LIN {X 0.008,Y -350.528,Z 1604.654,A 0.000,B 0.000,C 90.000,E1 117.719} C_DIS
LIN {X -0.132,Y -363.756,Z 1604.639,A 0.000,B 0.000,C 90.000,E1 115.027} C_DIS
LIN {X 0.133,Y -378.533,Z 1604.624,A 0.000,B 0.000,C 90.000,E1 112.333} C_DIS
LIN {X -0.125,Y -393.075,Z 1604.611,A 0.000,B 0.000,C 90.000,E1 110.066} C_DIS
LIN {X -0.167,Y -409.046,Z 1604.599,A 0.000,B 0.000,C 90.000,E1 107.819} C_DIS
LIN {X -0.066,Y -426.554,Z 1604.587,A 0.000,B 0.000,C 90.000,E1 105.607} C_DIS
LIN {X -0.040,Y -445.691,Z 1604.575,A 0.000,B 0.000,C 90.000,E1 103.467} C_DIS
LIN {X -0.108,Y -465.755,Z 1604.564,A 0.000,B 0.000,C 90.000,E1 101.478} C_DIS
LIN {X 0.275,Y -488.978,Z 1604.552,A 0.000,B 0.000,C 90.000,E1 99.378} C_DIS
LIN {X 0.186,Y -496.673,Z 1604.549,A 0.000,B 0.000,C 90.000,E1 98.746} C_DIS
LIN {X -0.096,Y -498.547,Z 1604.547,A 0.000,B 0.000,C 90.000,E1 98.568} C_DIS
LIN {X -0.248,Y -500.191,Z 1604.546,A 0.000,B 0.000,C 90.000,E1 98.341} C_DIS
LIN {X 0.168,Y -501.417,Z 1604.545,A 0.000,B 0.000,C 90.000,E1 98.049} C_DIS
LIN {X -0.044,Y -502.900,Z 1604.542,A 0.000,B 0.000,C 90.000,E1 97.587} C_DIS
LIN {X -0.248,Y -503.310,Z 1604.539,A 0.000,B 0.000,C 90.000,E1 97.125} C_DIS
LIN {X 0.057,Y -502.718,Z 1604.537,A 0.000,B 0.000,C 90.000,E1 96.606} C_DIS
LIN {X -0.137,Y -501.027,Z 1604.534,A 0.000,B 0.000,C 90.000,E1 96.144} C_DIS
LIN {X -0.208,Y -499.672,Z 1604.533,A 0.000,B 0.000,C 90.000,E1 95.910} C_DIS
LIN {X -0.198,Y -486.395,Z 1604.522,A 0.000,B 0.000,C 90.000,E1 93.955} C_DIS
LIN {X 0.123,Y -474.752,Z 1604.512,A 0.000,B 0.000,C 90.000,E1 92.178} C_DIS
LIN {X 0.139,Y -466.084,Z 1604.505,A 0.000,B 0.000,C 90.000,E1 90.917} C_DIS
LIN {X -0.196,Y -455.264,Z 1604.497,A 0.000,B 0.000,C 90.000,E1 89.427} C_DIS
LIN {X 0.202,Y -443.950,Z 1604.488,A 0.000,B 0.000,C 90.000,E1 87.822} C_DIS
LIN {X -0.200,Y -434.014,Z 1604.481,A 0.000,B 0.000,C 90.000,E1 86.560} C_DIS
LIN {X -0.045,Y -419.876,Z 1604.470,A 0.000,B 0.000,C 90.000,E1 84.666} C_DIS
LIN {X 0.148,Y -400.660,Z 1604.455,A 0.000,B 0.000,C 90.000,E1 81.894} C_DIS
LIN {X -0.093,Y -382.813,Z 1604.439,A 0.000,B 0.000,C 90.000,E1 79.106} C_DIS
LIN {X 0.129,Y -367.656,Z 1604.425,A 0.000,B 0.000,C 90.000,E1 76.464} C_DIS
LIN {X 0.070,Y -354.658,Z 1604.412,A 0.000,B 0.000,C 90.000,E1 74.102} C_DIS
LIN {X -0.105,Y -340.513,Z 1604.397,A 0.000,B 0.000,C 90.000,E1 71.402} C_DIS
LIN {X -0.038,Y -325.411,Z 1604.379,A 0.000,B 0.000,C 90.000,E1 68.284} C_DIS
LIN {X 0.018,Y -312.764,Z 1604.363,A 0.000,B 0.000,C 90.000,E1 65.409} C_DIS
LIN {X -0.037,Y -302.405,Z 1604.349,A 0.000,B 0.000,C 90.000,E1 62.820} C_DIS
LIN {X -0.068,Y -294.618,Z 1604.338,A 0.000,B 0.000,C 90.000,E1 60.845} C_DIS
LIN {X 0.011,Y -286.424,Z 1604.327,A 0.000,B 0.000,C 90.000,E1 58.820} C_DIS
LIN {X 0.017,Y -279.212,Z 1604.317,A 0.000,B 0.000,C 90.000,E1 57.120} C_DIS
LIN {X 0.002,Y -270.253,Z 1604.306,A 0.000,B 0.000,C 90.000,E1 55.055} C_DIS
LIN {X -0.130,Y -258.394,Z 1604.290,A 0.000,B 0.000,C 90.000,E1 52.271} C_DIS
LIN {X -0.056,Y -245.951,Z 1604.272,A 0.000,B 0.000,C 90.000,E1 49.013} C_DIS
LIN {X 0.127,Y -234.841,Z 1604.254,A 0.000,B 0.000,C 90.000,E1 45.648} C_DIS
LIN {X 0.000,Y -224.752,Z 1604.235,A 0.000,B 0.000,C 90.000,E1 42.285} C_DIS
LIN {X 0.071,Y -216.581,Z 1604.218,A 0.000,B 0.000,C 90.000,E1 39.197} C_DIS
LIN {X 0.010,Y -209.131,Z 1604.201,A 0.000,B 0.000,C 90.000,E1 36.091} C_DIS
LIN {X 0.035,Y -202.469,Z 1604.183,A 0.000,B 0.000,C 90.000,E1 32.911} C_DIS
LIN {X -0.046,Y -196.583,Z 1604.165,A 0.000,B 0.000,C 90.000,E1 29.716} C_DIS
LIN {X 0.024,Y -191.435,Z 1604.147,A 0.000,B 0.000,C 90.000,E1 26.437} C_DIS
LIN {X -0.020,Y -186.992,Z 1604.129,A 0.000,B 0.000,C 90.000,E1 23.153} C_DIS
LIN {X 0.069,Y -182.336,Z 1604.105,A 0.000,B 0.000,C 90.000,E1 18.960} C_DIS
LIN {X 0.001,Y -178.430,Z 1604.082,A 0.000,B 0.000,C 90.000,E1 14.773} C_DIS
LIN {X 0.016,Y -174.791,Z 1604.054,A 0.000,B 0.000,C 90.000,E1 9.670} C_DIS
LIN {X 0.026,Y -172.085,Z 1604.020,A 0.000,B 0.000,C 90.000,E1 3.669} C_DIS
LIN {X 0.012,Y -172.894,Z 1603.926,A 0.000,B 0.000,C 90.000,E1 346.589} C_DIS
LIN {X -0.013,Y -175.478,Z 1603.902,A 0.000,B 0.000,C 90.000,E1 342.308} C_DIS
LIN {X -0.027,Y -178.547,Z 1603.883,A 0.000,B 0.000,C 90.000,E1 338.901} C_DIS
LIN {X 0.066,Y -182.394,Z 1603.864,A 0.000,B 0.000,C 90.000,E1 335.485} C_DIS
LIN {X -0.013,Y -186.994,Z 1603.845,A 0.000,B 0.000,C 90.000,E1 332.153} C_DIS
LIN {X 0.030,Y -192.401,Z 1603.827,A 0.000,B 0.000,C 90.000,E1 328.820} C_DIS
LIN {X 0.008,Y -198.593,Z 1603.809,A 0.000,B 0.000,C 90.000,E1 325.548} C_DIS
LIN {X -0.001,Y -205.535,Z 1603.791,A 0.000,B 0.000,C 90.000,E1 322.316} C_DIS
LIN {X -0.016,Y -213.403,Z 1603.773,A 0.000,B 0.000,C 90.000,E1 319.138} C_DIS
LIN {X 0.146,Y -222.186,Z 1603.756,A 0.000,B 0.000,C 90.000,E1 315.972} C_DIS
LIN {X 0.053,Y -231.907,Z 1603.739,A 0.000,B 0.000,C 90.000,E1 312.933} C_DIS
LIN {X -0.073,Y -241.420,Z 1603.724,A 0.000,B 0.000,C 90.000,E1 310.334} C_DIS
LIN {X 0.026,Y -249.142,Z 1603.714,A 0.000,B 0.000,C 90.000,E1 308.463} C_DIS
LIN {X -0.056,Y -257.815,Z 1603.704,A 0.000,B 0.000,C 90.000,E1 306.664} C_DIS
LIN {X -0.011,Y -267.503,Z 1603.694,A 0.000,B 0.000,C 90.000,E1 304.865} C_DIS
LIN {X -0.002,Y -282.651,Z 1603.680,A 0.000,B 0.000,C 90.000,E1 302.418} C_DIS
LIN {X -0.183,Y -304.189,Z 1603.663,A 0.000,B 0.000,C 90.000,E1 299.411} C_DIS
LIN {X 0.112,Y -316.699,Z 1603.654,A 0.000,B 0.000,C 90.000,E1 297.719} C_DIS
LIN {X 0.182,Y -329.058,Z 1603.645,A 0.000,B 0.000,C 90.000,E1 296.104} C_DIS
LIN {X -0.139,Y -341.231,Z 1603.636,A 0.000,B 0.000,C 90.000,E1 294.591} C_DIS
LIN {X -0.183,Y -360.570,Z 1603.623,A 0.000,B 0.000,C 90.000,E1 292.153} C_DIS
LIN {X 0.161,Y -372.793,Z 1603.615,A 0.000,B 0.000,C 90.000,E1 290.610} C_DIS
LIN {X -0.012,Y -379.855,Z 1603.610,A 0.000,B 0.000,C 90.000,E1 289.758} C_DIS
LIN {X -0.133,Y -386.447,Z 1603.605,A 0.000,B 0.000,C 90.000,E1 288.906} C_DIS
LIN {X -0.157,Y -394.469,Z 1603.599,A 0.000,B 0.000,C 90.000,E1 287.764} C_DIS
LIN {X -0.143,Y -399.824,Z 1603.594,A 0.000,B 0.000,C 90.000,E1 286.913} C_DIS
LIN {X 0.183,Y -404.463,Z 1603.589,A 0.000,B 0.000,C 90.000,E1 286.024} C_DIS
LIN {X 0.078,Y -407.037,Z 1603.586,A 0.000,B 0.000,C 90.000,E1 285.481} C_DIS
LIN {X -0.122,Y -409.192,Z 1603.583,A 0.000,B 0.000,C 90.000,E1 284.954} C_DIS
LIN {X 0.194,Y -410.983,Z 1603.580,A 0.000,B 0.000,C 90.000,E1 284.356} C_DIS
LIN {X 0.017,Y -412.380,Z 1603.577,A 0.000,B 0.000,C 90.000,E1 283.828} C_DIS
LIN {X -0.150,Y -413.367,Z 1603.574,A 0.000,B 0.000,C 90.000,E1 283.300} C_DIS
LIN {X 0.096,Y -413.834,Z 1603.571,A 0.000,B 0.000,C 90.000,E1 282.715} C_DIS
LIN {X -0.054,Y -413.863,Z 1603.568,A 0.000,B 0.000,C 90.000,E1 282.187} C_DIS
LIN {X -0.202,Y -413.406,Z 1603.565,A 0.000,B 0.000,C 90.000,E1 281.658} C_DIS
LIN {X 0.055,Y -412.391,Z 1603.562,A 0.000,B 0.000,C 90.000,E1 281.074} C_DIS
LIN {X -0.097,Y -410.846,Z 1603.558,A 0.000,B 0.000,C 90.000,E1 280.546} C_DIS
LIN {X 0.146,Y -408.639,Z 1603.555,A 0.000,B 0.000,C 90.000,E1 279.962} C_DIS
LIN {X -0.096,Y -405.779,Z 1603.552,A 0.000,B 0.000,C 90.000,E1 279.443} C_DIS
LIN {X 0.112,Y -402.193,Z 1603.549,A 0.000,B 0.000,C 90.000,E1 278.859} C_DIS
LIN {X -0.156,Y -397.944,Z 1603.546,A 0.000,B 0.000,C 90.000,E1 278.341} C_DIS
LIN {X 0.004,Y -393.129,Z 1603.543,A 0.000,B 0.000,C 90.000,E1 277.757} C_DIS
LIN {X 0.079,Y -387.589,Z 1603.540,A 0.000,B 0.000,C 90.000,E1 277.182} C_DIS
LIN {X -0.008,Y -381.681,Z 1603.537,A 0.000,B 0.000,C 90.000,E1 276.663} C_DIS
LIN {X -0.152,Y -375.722,Z 1603.534,A 0.000,B 0.000,C 90.000,E1 276.201} C_DIS
LIN {X -0.050,Y -369.564,Z 1603.532,A 0.000,B 0.000,C 90.000,E1 275.739} C_DIS
LIN {X -0.163,Y -360.209,Z 1603.529,A 0.000,B 0.000,C 90.000,E1 275.163} C_DIS
LIN {X 0.105,Y -350.532,Z 1603.526,A 0.000,B 0.000,C 90.000,E1 274.588} C_DIS
LIN {X 0.036,Y -340.918,Z 1603.523,A 0.000,B 0.000,C 90.000,E1 274.131} C_DIS
LIN {X -0.123,Y -331.187,Z 1603.521,A 0.000,B 0.000,C 90.000,E1 273.726} C_DIS
LIN {X -0.084,Y -321.122,Z 1603.518,A 0.000,B 0.000,C 90.000,E1 273.326} C_DIS
LIN {X -0.118,Y -310.846,Z 1603.516,A 0.000,B 0.000,C 90.000,E1 272.980} C_DIS
LIN {X 0.130,Y -300.673,Z 1603.515,A 0.000,B 0.000,C 90.000,E1 272.636} C_DIS
LIN {X 0.110,Y -293.452,Z 1603.514,A 0.000,B 0.000,C 90.000,E1 272.465} C_DIS
LIN {X -0.070,Y -285.552,Z 1603.513,A 0.000,B 0.000,C 90.000,E1 272.350} C_DIS
LIN {X -0.105,Y -271.786,Z 1603.512,A 0.000,B 0.000,C 90.000,E1 272.178} C_DIS
LIN {X 0.049,Y -251.939,Z 1603.511,A 0.000,B 0.000,C 90.000,E1 271.949} C_DIS
LIN {X 0.003,Y -228.720,Z 1603.510,A 0.000,B 0.000,C 90.000,E1 271.835} C_DIS
LIN {X -0.037,Y -219.677,Z 1603.510,A 0.000,B 0.000,C 90.000,E1 271.835} C_DIS
LIN {X -0.064,Y -181.293,Z 1603.510,A 0.000,B 0.000,C 90.000,E1 271.835} C_DIS
LIN {X -0.052,Y -181.573,Z 1603.500,A 0.000,B 0.000,C 90.000,E1 270.115} C_DIS
LIN {X -0.064,Y -180.871,Z 1603.472,A 0.000,B 0.000,C 90.000,E1 265.065} C_DIS
LIN {X -0.007,Y -178.987,Z 1603.444,A 0.000,B 0.000,C 90.000,E1 259.982} C_DIS
LIN {X 0.004,Y -177.968,Z 1603.435,A 0.000,B 0.000,C 90.000,E1 258.285} C_DIS
LIN {X 0.023,Y -175.612,Z 1603.411,A 0.000,B 0.000,C 90.000,E1 254.031} C_DIS
LIN {X 0.035,Y -172.333,Z 1603.388,A 0.000,B 0.000,C 90.000,E1 249.752} C_DIS
LIN {X 0.014,Y -171.810,Z 1603.383,A 0.000,B 0.000,C 90.000,E1 248.901} C_DIS
LIN {X 0.021,Y -170.273,Z 1603.373,A 0.000,B 0.000,C 90.000,E1 247.177} C_DIS
LIN {X -0.043,Y -166.814,Z 1603.349,A 0.000,B 0.000,C 90.000,E1 242.871} C_DIS
LIN {X 0.015,Y -162.795,Z 1603.325,A 0.000,B 0.000,C 90.000,E1 238.486} C_DIS
LIN {X 0.074,Y -161.483,Z 1603.315,A 0.000,B 0.000,C 90.000,E1 236.707} C_DIS
LIN {X -0.009,Y -157.479,Z 1603.291,A 0.000,B 0.000,C 90.000,E1 232.316} C_DIS
LIN {X 0.048,Y -155.495,Z 1603.276,A 0.000,B 0.000,C 90.000,E1 229.622} C_DIS
LIN {X -0.021,Y -151.801,Z 1603.251,A 0.000,B 0.000,C 90.000,E1 225.162} C_DIS
LIN {X -0.008,Y -150.011,Z 1603.236,A 0.000,B 0.000,C 90.000,E1 222.447} C_DIS
LIN {X 0.023,Y -146.835,Z 1603.211,A 0.000,B 0.000,C 90.000,E1 217.890} C_DIS
LIN {X 0.010,Y -145.417,Z 1603.195,A 0.000,B 0.000,C 90.000,E1 215.152} C_DIS
LIN {X 0.045,Y -142.846,Z 1603.170,A 0.000,B 0.000,C 90.000,E1 210.541} C_DIS
LIN {X -0.024,Y -141.460,Z 1603.149,A 0.000,B 0.000,C 90.000,E1 206.873} C_DIS
LIN {X 0.015,Y -139.374,Z 1603.113,A 0.000,B 0.000,C 90.000,E1 200.355} C_DIS
LIN {X -0.043,Y -138.825,Z 1603.098,A 0.000,B 0.000,C 90.000,E1 197.583} C_DIS
LIN {X 0.045,Y -138.353,Z 1603.056,A 0.000,B 0.000,C 90.000,E1 190.074} C_DIS
LIN {X 0.019,Y -139.531,Z 1603.004,A 0.000,B 0.000,C 90.000,E1 180.745} C_DIS
LIN {X -0.029,Y -141.210,Z 1602.973,A 0.000,B 0.000,C 90.000,E1 175.179} C_DIS
LIN {X 0.072,Y -142.584,Z 1602.958,A 0.000,B 0.000,C 90.000,E1 172.356} C_DIS
LIN {X 0.025,Y -144.881,Z 1602.932,A 0.000,B 0.000,C 90.000,E1 167.757} C_DIS
LIN {X -0.020,Y -147.508,Z 1602.912,A 0.000,B 0.000,C 90.000,E1 164.102} C_DIS
LIN {X 0.054,Y -150.101,Z 1602.891,A 0.000,B 0.000,C 90.000,E1 160.423} C_DIS
LIN {X 0.067,Y -153.457,Z 1602.871,A 0.000,B 0.000,C 90.000,E1 156.794} C_DIS
LIN {X -0.081,Y -157.821,Z 1602.846,A 0.000,B 0.000,C 90.000,E1 152.359} C_DIS
LIN {X -0.050,Y -162.104,Z 1602.827,A 0.000,B 0.000,C 90.000,E1 148.791} C_DIS
LIN {X -0.026,Y -166.305,Z 1602.807,A 0.000,B 0.000,C 90.000,E1 145.261} C_DIS
LIN {X -0.029,Y -171.321,Z 1602.788,A 0.000,B 0.000,C 90.000,E1 141.778} C_DIS
LIN {X 0.005,Y -176.221,Z 1602.768,A 0.000,B 0.000,C 90.000,E1 138.324} C_DIS
LIN {X -0.001,Y -180.500,Z 1602.754,A 0.000,B 0.000,C 90.000,E1 135.769} C_DIS
LIN {X -0.020,Y -185.903,Z 1602.736,A 0.000,B 0.000,C 90.000,E1 132.405} C_DIS
LIN {X 0.041,Y -190.530,Z 1602.722,A 0.000,B 0.000,C 90.000,E1 129.886} C_DIS
LIN {X 0.072,Y -196.281,Z 1602.703,A 0.000,B 0.000,C 90.000,E1 126.583} C_DIS
LIN {X -0.128,Y -201.084,Z 1602.690,A 0.000,B 0.000,C 90.000,E1 124.199} C_DIS
LIN {X 0.041,Y -205.074,Z 1602.677,A 0.000,B 0.000,C 90.000,E1 121.926} C_DIS
LIN {X 0.030,Y -323.152,Z 1602.677,A 0.000,B 0.000,C 90.000,E1 121.926} C_DIS
LIN {X -0.040,Y -324.187,Z 1602.677,A 0.000,B 0.000,C 90.000,E1 121.926} C_DIS
LIN {X -0.029,Y -328.842,Z 1602.676,A 0.000,B 0.000,C 90.000,E1 121.750} C_DIS
LIN {X -0.017,Y -331.941,Z 1602.675,A 0.000,B 0.000,C 90.000,E1 121.514} C_DIS
LIN {X 0.089,Y -335.653,Z 1602.673,A 0.000,B 0.000,C 90.000,E1 121.052} C_DIS
LIN {X 0.042,Y -337.481,Z 1602.671,A 0.000,B 0.000,C 90.000,E1 120.747} C_DIS
LIN {X 0.163,Y -341.409,Z 1602.666,A 0.000,B 0.000,C 90.000,E1 119.795} C_DIS
LIN {X -0.067,Y -353.529,Z 1602.650,A 0.000,B 0.000,C 90.000,E1 117.078} C_DIS
LIN {X -0.127,Y -367.117,Z 1602.635,A 0.000,B 0.000,C 90.000,E1 114.387} C_DIS
LIN {X -0.040,Y -380.518,Z 1602.622,A 0.000,B 0.000,C 90.000,E1 112.025} C_DIS
LIN {X 0.115,Y -395.258,Z 1602.610,A 0.000,B 0.000,C 90.000,E1 109.704} C_DIS
LIN {X 0.137,Y -411.443,Z 1602.597,A 0.000,B 0.000,C 90.000,E1 107.457} C_DIS
LIN {X -0.105,Y -429.183,Z 1602.585,A 0.000,B 0.000,C 90.000,E1 105.300} C_DIS
LIN {X -0.098,Y -448.526,Z 1602.573,A 0.000,B 0.000,C 90.000,E1 103.175} C_DIS
LIN {X 0.031,Y -468.673,Z 1602.562,A 0.000,B 0.000,C 90.000,E1 101.186} C_DIS
LIN {X 0.086,Y -491.952,Z 1602.551,A 0.000,B 0.000,C 90.000,E1 99.151} C_DIS
LIN {X -0.093,Y -496.937,Z 1602.549,A 0.000,B 0.000,C 90.000,E1 98.746} C_DIS
LIN {X 0.120,Y -498.714,Z 1602.547,A 0.000,B 0.000,C 90.000,E1 98.511} C_DIS
LIN {X 0.041,Y -500.280,Z 1602.546,A 0.000,B 0.000,C 90.000,E1 98.276} C_DIS
LIN {X -0.110,Y -501.446,Z 1602.545,A 0.000,B 0.000,C 90.000,E1 98.049} C_DIS
LIN {X 0.178,Y -502.831,Z 1602.542,A 0.000,B 0.000,C 90.000,E1 97.530} C_DIS
LIN {X -0.026,Y -503.158,Z 1602.539,A 0.000,B 0.000,C 90.000,E1 97.068} C_DIS
LIN {X -0.221,Y -502.481,Z 1602.537,A 0.000,B 0.000,C 90.000,E1 96.606} C_DIS
LIN {X 0.084,Y -500.688,Z 1602.534,A 0.000,B 0.000,C 90.000,E1 96.087} C_DIS
LIN {X 0.011,Y -499.267,Z 1602.532,A 0.000,B 0.000,C 90.000,E1 95.853} C_DIS
LIN {X 0.008,Y -485.988,Z 1602.522,A 0.000,B 0.000,C 90.000,E1 93.898} C_DIS
LIN {X -0.158,Y -474.365,Z 1602.512,A 0.000,B 0.000,C 90.000,E1 92.178} C_DIS
LIN {X -0.141,Y -465.703,Z 1602.505,A 0.000,B 0.000,C 90.000,E1 90.917} C_DIS
LIN {X -0.020,Y -454.847,Z 1602.496,A 0.000,B 0.000,C 90.000,E1 89.370} C_DIS
LIN {X 0.172,Y -445.458,Z 1602.489,A 0.000,B 0.000,C 90.000,E1 88.051} C_DIS
LIN {X 0.223,Y -435.595,Z 1602.482,A 0.000,B 0.000,C 90.000,E1 86.731} C_DIS
LIN {X -0.014,Y -421.453,Z 1602.472,A 0.000,B 0.000,C 90.000,E1 84.894} C_DIS
LIN {X -0.131,Y -400.261,Z 1602.455,A 0.000,B 0.000,C 90.000,E1 81.894} C_DIS
LIN {X 0.005,Y -382.444,Z 1602.439,A 0.000,B 0.000,C 90.000,E1 79.050} C_DIS
LIN {X -0.147,Y -367.291,Z 1602.425,A 0.000,B 0.000,C 90.000,E1 76.464} C_DIS
LIN {X -0.206,Y -354.309,Z 1602.411,A 0.000,B 0.000,C 90.000,E1 74.102} C_DIS
LIN {X 0.052,Y -340.157,Z 1602.396,A 0.000,B 0.000,C 90.000,E1 71.329} C_DIS
LIN {X -0.008,Y -325.083,Z 1602.379,A 0.000,B 0.000,C 90.000,E1 68.230} C_DIS
LIN {X 0.032,Y -312.431,Z 1602.363,A 0.000,B 0.000,C 90.000,E1 65.357} C_DIS
LIN {X 0.098,Y -302.029,Z 1602.349,A 0.000,B 0.000,C 90.000,E1 62.743} C_DIS
LIN {X -0.081,Y -294.205,Z 1602.338,A 0.000,B 0.000,C 90.000,E1 60.795} C_DIS
LIN {X 0.132,Y -285.978,Z 1602.327,A 0.000,B 0.000,C 90.000,E1 58.742} C_DIS
LIN {X 0.132,Y -278.724,Z 1602.317,A 0.000,B 0.000,C 90.000,E1 57.041} C_DIS
LIN {X 0.107,Y -269.761,Z 1602.306,A 0.000,B 0.000,C 90.000,E1 54.975} C_DIS
LIN {X 0.010,Y -256.519,Z 1602.288,A 0.000,B 0.000,C 90.000,E1 51.823} C_DIS
LIN {X 0.023,Y -244.339,Z 1602.270,A 0.000,B 0.000,C 90.000,E1 48.566} C_DIS
LIN {X -0.009,Y -233.391,Z 1602.251,A 0.000,B 0.000,C 90.000,E1 45.243} C_DIS
LIN {X 0.055,Y -224.511,Z 1602.234,A 0.000,B 0.000,C 90.000,E1 42.204} C_DIS
LIN {X 0.117,Y -216.388,Z 1602.218,A 0.000,B 0.000,C 90.000,E1 39.116} C_DIS
LIN {X 0.047,Y -208.969,Z 1602.200,A 0.000,B 0.000,C 90.000,E1 36.011} C_DIS
LIN {X 0.065,Y -202.346,Z 1602.182,A 0.000,B 0.000,C 90.000,E1 32.832} C_DIS
LIN {X 0.050,Y -196.497,Z 1602.165,A 0.000,B 0.000,C 90.000,E1 29.617} C_DIS
LIN {X 0.039,Y -191.390,Z 1602.146,A 0.000,B 0.000,C 90.000,E1 26.360} C_DIS
LIN {X -0.011,Y -186.993,Z 1602.128,A 0.000,B 0.000,C 90.000,E1 23.078} C_DIS
LIN {X 0.010,Y -182.370,Z 1602.105,A 0.000,B 0.000,C 90.000,E1 18.906} C_DIS
LIN {X -0.051,Y -178.501,Z 1602.082,A 0.000,B 0.000,C 90.000,E1 14.717} C_DIS
LIN {X -0.029,Y -174.893,Z 1602.053,A 0.000,B 0.000,C 90.000,E1 9.613} C_DIS
LIN {X -0.011,Y -172.248,Z 1602.020,A 0.000,B 0.000,C 90.000,E1 3.612} C_DIS
LIN {X 0.031,Y -173.129,Z 1601.926,A 0.000,B 0.000,C 90.000,E1 346.589} C_DIS
LIN {X 0.013,Y -175.709,Z 1601.902,A 0.000,B 0.000,C 90.000,E1 342.308} C_DIS
LIN {X 0.006,Y -178.767,Z 1601.883,A 0.000,B 0.000,C 90.000,E1 338.901} C_DIS
LIN {X -0.062,Y -182.613,Z 1601.864,A 0.000,B 0.000,C 90.000,E1 335.537} C_DIS
LIN {X 0.033,Y -187.197,Z 1601.845,A 0.000,B 0.000,C 90.000,E1 332.153} C_DIS
LIN {X -0.083,Y -192.573,Z 1601.827,A 0.000,B 0.000,C 90.000,E1 328.869} C_DIS
LIN {X -0.098,Y -198.723,Z 1601.809,A 0.000,B 0.000,C 90.000,E1 325.595} C_DIS
LIN {X -0.064,Y -205.638,Z 1601.791,A 0.000,B 0.000,C 90.000,E1 322.351} C_DIS
LIN {X 0.051,Y -213.470,Z 1601.773,A 0.000,B 0.000,C 90.000,E1 319.138} C_DIS
LIN {X -0.096,Y -222.212,Z 1601.756,A 0.000,B 0.000,C 90.000,E1 316.053} C_DIS
LIN {X -0.042,Y -231.891,Z 1601.739,A 0.000,B 0.000,C 90.000,E1 312.975} C_DIS
LIN {X 0.004,Y -241.330,Z 1601.724,A 0.000,B 0.000,C 90.000,E1 310.334} C_DIS
LIN {X 0.104,Y -249.003,Z 1601.714,A 0.000,B 0.000,C 90.000,E1 308.463} C_DIS
LIN {X 0.022,Y -257.648,Z 1601.704,A 0.000,B 0.000,C 90.000,E1 306.664} C_DIS
LIN {X -0.085,Y -267.352,Z 1601.694,A 0.000,B 0.000,C 90.000,E1 304.898} C_DIS
LIN {X 0.079,Y -282.490,Z 1601.680,A 0.000,B 0.000,C 90.000,E1 302.418} C_DIS
LIN {X -0.102,Y -304.049,Z 1601.663,A 0.000,B 0.000,C 90.000,E1 299.411} C_DIS
LIN {X -0.086,Y -316.547,Z 1601.654,A 0.000,B 0.000,C 90.000,E1 297.769} C_DIS
LIN {X -0.029,Y -328.899,Z 1601.645,A 0.000,B 0.000,C 90.000,E1 296.155} C_DIS
LIN {X -0.055,Y -341.097,Z 1601.637,A 0.000,B 0.000,C 90.000,E1 294.591} C_DIS
LIN {X -0.089,Y -360.452,Z 1601.623,A 0.000,B 0.000,C 90.000,E1 292.153} C_DIS
LIN {X 0.013,Y -375.109,Z 1601.613,A 0.000,B 0.000,C 90.000,E1 290.355} C_DIS
LIN {X 0.207,Y -382.083,Z 1601.608,A 0.000,B 0.000,C 90.000,E1 289.450} C_DIS
LIN {X 0.115,Y -388.538,Z 1601.603,A 0.000,B 0.000,C 90.000,E1 288.598} C_DIS
LIN {X -0.048,Y -394.507,Z 1601.599,A 0.000,B 0.000,C 90.000,E1 287.764} C_DIS
LIN {X -0.033,Y -399.917,Z 1601.594,A 0.000,B 0.000,C 90.000,E1 286.913} C_DIS
LIN {X 0.219,Y -403.151,Z 1601.591,A 0.000,B 0.000,C 90.000,E1 286.315} C_DIS
LIN {X -0.006,Y -405.978,Z 1601.588,A 0.000,B 0.000,C 90.000,E1 285.788} C_DIS
LIN {X -0.006,Y -409.395,Z 1601.583,A 0.000,B 0.000,C 90.000,E1 284.954} C_DIS
LIN {X -0.086,Y -411.232,Z 1601.580,A 0.000,B 0.000,C 90.000,E1 284.411} C_DIS
LIN {X 0.136,Y -412.650,Z 1601.577,A 0.000,B 0.000,C 90.000,E1 283.828} C_DIS
LIN {X -0.030,Y -413.653,Z 1601.574,A 0.000,B 0.000,C 90.000,E1 283.300} C_DIS
LIN {X -0.185,Y -414.163,Z 1601.571,A 0.000,B 0.000,C 90.000,E1 282.771} C_DIS
LIN {X 0.070,Y -414.229,Z 1601.568,A 0.000,B 0.000,C 90.000,E1 282.187} C_DIS
LIN {X -0.076,Y -413.772,Z 1601.565,A 0.000,B 0.000,C 90.000,E1 281.658} C_DIS
LIN {X -0.222,Y -412.853,Z 1601.562,A 0.000,B 0.000,C 90.000,E1 281.130} C_DIS
LIN {X 0.032,Y -411.338,Z 1601.559,A 0.000,B 0.000,C 90.000,E1 280.546} C_DIS
LIN {X -0.124,Y -409.180,Z 1601.556,A 0.000,B 0.000,C 90.000,E1 280.018} C_DIS
LIN {X 0.043,Y -406.361,Z 1601.552,A 0.000,B 0.000,C 90.000,E1 279.443} C_DIS
LIN {X -0.143,Y -402.813,Z 1601.549,A 0.000,B 0.000,C 90.000,E1 278.916} C_DIS
LIN {X -0.013,Y -398.578,Z 1601.546,A 0.000,B 0.000,C 90.000,E1 278.341} C_DIS
LIN {X 0.149,Y -393.758,Z 1601.543,A 0.000,B 0.000,C 90.000,E1 277.757} C_DIS
LIN {X -0.158,Y -388.263,Z 1601.540,A 0.000,B 0.000,C 90.000,E1 277.239} C_DIS
LIN {X 0.135,Y -382.377,Z 1601.537,A 0.000,B 0.000,C 90.000,E1 276.663} C_DIS
LIN {X 0.054,Y -373.456,Z 1601.533,A 0.000,B 0.000,C 90.000,E1 275.967} C_DIS
LIN {X -0.123,Y -367.213,Z 1601.531,A 0.000,B 0.000,C 90.000,E1 275.568} C_DIS
LIN {X -0.021,Y -360.942,Z 1601.529,A 0.000,B 0.000,C 90.000,E1 275.163} C_DIS
LIN {X -0.073,Y -351.359,Z 1601.526,A 0.000,B 0.000,C 90.000,E1 274.645} C_DIS
LIN {X -0.151,Y -341.632,Z 1601.523,A 0.000,B 0.000,C 90.000,E1 274.188} C_DIS
LIN {X 0.034,Y -331.902,Z 1601.521,A 0.000,B 0.000,C 90.000,E1 273.726} C_DIS
LIN {X 0.093,Y -322.069,Z 1601.519,A 0.000,B 0.000,C 90.000,E1 273.326} C_DIS
LIN {X 0.047,Y -311.873,Z 1601.517,A 0.000,B 0.000,C 90.000,E1 272.980} C_DIS
LIN {X -0.029,Y -301.793,Z 1601.515,A 0.000,B 0.000,C 90.000,E1 272.694} C_DIS
LIN {X 0.132,Y -290.807,Z 1601.514,A 0.000,B 0.000,C 90.000,E1 272.407} C_DIS
LIN {X -0.028,Y -282.233,Z 1601.513,A 0.000,B 0.000,C 90.000,E1 272.293} C_DIS
LIN {X 0.062,Y -258.479,Z 1601.511,A 0.000,B 0.000,C 90.000,E1 272.007} C_DIS
LIN {X 0.037,Y -241.854,Z 1601.511,A 0.000,B 0.000,C 90.000,E1 271.892} C_DIS
LIN {X 0.045,Y -228.495,Z 1601.510,A 0.000,B 0.000,C 90.000,E1 271.835} C_DIS
LIN {X 0.002,Y -181.289,Z 1601.510,A 0.000,B 0.000,C 90.000,E1 271.835} C_DIS
LIN {X -0.018,Y -181.574,Z 1601.501,A 0.000,B 0.000,C 90.000,E1 270.115} C_DIS
LIN {X -0.030,Y -180.873,Z 1601.473,A 0.000,B 0.000,C 90.000,E1 265.065} C_DIS
LIN {X 0.026,Y -178.990,Z 1601.444,A 0.000,B 0.000,C 90.000,E1 259.982} C_DIS
LIN {X 0.037,Y -177.975,Z 1601.435,A 0.000,B 0.000,C 90.000,E1 258.285} C_DIS
LIN {X 0.056,Y -175.619,Z 1601.411,A 0.000,B 0.000,C 90.000,E1 254.031} C_DIS
LIN {X 0.068,Y -172.340,Z 1601.388,A 0.000,B 0.000,C 90.000,E1 249.752} C_DIS
LIN {X 0.046,Y -171.816,Z 1601.383,A 0.000,B 0.000,C 90.000,E1 248.901} C_DIS
LIN {X 0.053,Y -170.283,Z 1601.373,A 0.000,B 0.000,C 90.000,E1 247.177} C_DIS
LIN {X -0.011,Y -166.822,Z 1601.349,A 0.000,B 0.000,C 90.000,E1 242.871} C_DIS
LIN {X -0.092,Y -162.805,Z 1601.325,A 0.000,B 0.000,C 90.000,E1 238.535} C_DIS
LIN {X -0.029,Y -161.491,Z 1601.315,A 0.000,B 0.000,C 90.000,E1 236.755} C_DIS
LIN {X 0.021,Y -157.488,Z 1601.291,A 0.000,B 0.000,C 90.000,E1 232.316} C_DIS
LIN {X -0.040,Y -155.506,Z 1601.276,A 0.000,B 0.000,C 90.000,E1 229.666} C_DIS
LIN {X 0.010,Y -151.809,Z 1601.251,A 0.000,B 0.000,C 90.000,E1 225.162} C_DIS
LIN {X 0.023,Y -150.021,Z 1601.236,A 0.000,B 0.000,C 90.000,E1 222.447} C_DIS
LIN {X 0.053,Y -146.842,Z 1601.211,A 0.000,B 0.000,C 90.000,E1 217.890} C_DIS
LIN {X -0.044,Y -145.424,Z 1601.195,A 0.000,B 0.000,C 90.000,E1 215.185} C_DIS
LIN {X -0.048,Y -142.851,Z 1601.170,A 0.000,B 0.000,C 90.000,E1 210.590} C_DIS
LIN {X 0.004,Y -141.465,Z 1601.149,A 0.000,B 0.000,C 90.000,E1 206.873} C_DIS
LIN {X -0.005,Y -139.376,Z 1601.113,A 0.000,B 0.000,C 90.000,E1 200.375} C_DIS
LIN {X -0.014,Y -138.828,Z 1601.098,A 0.000,B 0.000,C 90.000,E1 197.583} C_DIS
LIN {X 0.050,Y -138.353,Z 1601.056,A 0.000,B 0.000,C 90.000,E1 190.084} C_DIS
LIN {X 0.047,Y -139.528,Z 1601.004,A 0.000,B 0.000,C 90.000,E1 180.745} C_DIS
LIN {X 0.001,Y -141.204,Z 1600.973,A 0.000,B 0.000,C 90.000,E1 175.179} C_DIS
LIN {X -0.040,Y -142.580,Z 1600.958,A 0.000,B 0.000,C 90.000,E1 172.413} C_DIS
LIN {X 0.056,Y -144.874,Z 1600.932,A 0.000,B 0.000,C 90.000,E1 167.757} C_DIS
LIN {X 0.010,Y -147.500,Z 1600.912,A 0.000,B 0.000,C 90.000,E1 164.102} C_DIS
LIN {X 0.085,Y -150.091,Z 1600.891,A 0.000,B 0.000,C 90.000,E1 160.423} C_DIS
LIN {X -0.044,Y -153.445,Z 1600.871,A 0.000,B 0.000,C 90.000,E1 156.847} C_DIS
LIN {X -0.051,Y -157.808,Z 1600.846,A 0.000,B 0.000,C 90.000,E1 152.359} C_DIS
LIN {X -0.018,Y -162.090,Z 1600.827,A 0.000,B 0.000,C 90.000,E1 148.791} C_DIS
LIN {X 0.007,Y -166.290,Z 1600.807,A 0.000,B 0.000,C 90.000,E1 145.261} C_DIS
LIN {X 0.004,Y -171.307,Z 1600.788,A 0.000,B 0.000,C 90.000,E1 141.778} C_DIS
LIN {X 0.039,Y -176.204,Z 1600.769,A 0.000,B 0.000,C 90.000,E1 138.324} C_DIS
LIN {X -0.096,Y -180.480,Z 1600.754,A 0.000,B 0.000,C 90.000,E1 135.810} C_DIS
LIN {X 0.015,Y -185.885,Z 1600.736,A 0.000,B 0.000,C 90.000,E1 132.405} C_DIS
LIN {X -0.070,Y -190.510,Z 1600.722,A 0.000,B 0.000,C 90.000,E1 129.930} C_DIS
LIN {X 0.108,Y -196.261,Z 1600.703,A 0.000,B 0.000,C 90.000,E1 126.583} C_DIS
LIN {X -0.092,Y -201.066,Z 1600.690,A 0.000,B 0.000,C 90.000,E1 124.199} C_DIS
LIN {X -0.113,Y -205.005,Z 1600.678,A 0.000,B 0.000,C 90.000,E1 122.005} C_DIS
LIN {X 0.062,Y -323.204,Z 1600.678,A 0.000,B 0.000,C 90.000,E1 121.957} C_DIS
LIN {X -0.009,Y -324.124,Z 1600.677,A 0.000,B 0.000,C 90.000,E1 121.957} C_DIS
LIN {X 0.030,Y -329.117,Z 1600.676,A 0.000,B 0.000,C 90.000,E1 121.750} C_DIS
LIN {X -0.047,Y -332.218,Z 1600.675,A 0.000,B 0.000,C 90.000,E1 121.514} C_DIS
LIN {X -0.082,Y -335.915,Z 1600.672,A 0.000,B 0.000,C 90.000,E1 121.052} C_DIS
LIN {X 0.042,Y -337.643,Z 1600.671,A 0.000,B 0.000,C 90.000,E1 120.718} C_DIS
LIN {X 0.045,Y -352.222,Z 1600.652,A 0.000,B 0.000,C 90.000,E1 117.334} C_DIS
LIN {X -0.040,Y -365.654,Z 1600.637,A 0.000,B 0.000,C 90.000,E1 114.643} C_DIS
LIN {X 0.131,Y -380.659,Z 1600.622,A 0.000,B 0.000,C 90.000,E1 111.972} C_DIS
LIN {X 0.064,Y -395.416,Z 1600.609,A 0.000,B 0.000,C 90.000,E1 109.685} C_DIS
LIN {X -0.051,Y -411.618,Z 1600.597,A 0.000,B 0.000,C 90.000,E1 107.457} C_DIS
LIN {X 0.116,Y -429.376,Z 1600.585,A 0.000,B 0.000,C 90.000,E1 105.245} C_DIS
LIN {X 0.148,Y -448.734,Z 1600.573,A 0.000,B 0.000,C 90.000,E1 103.119} C_DIS
LIN {X -0.153,Y -468.887,Z 1600.562,A 0.000,B 0.000,C 90.000,E1 101.186} C_DIS
LIN {X -0.091,Y -492.172,Z 1600.551,A 0.000,B 0.000,C 90.000,E1 99.151} C_DIS
LIN {X 0.085,Y -494.812,Z 1600.550,A 0.000,B 0.000,C 90.000,E1 98.916} C_DIS
LIN {X -0.268,Y -497.071,Z 1600.548,A 0.000,B 0.000,C 90.000,E1 98.746} C_DIS
LIN {X -0.056,Y -498.785,Z 1600.547,A 0.000,B 0.000,C 90.000,E1 98.511} C_DIS
LIN {X -0.134,Y -500.298,Z 1600.546,A 0.000,B 0.000,C 90.000,E1 98.276} C_DIS
LIN {X 0.211,Y -501.421,Z 1600.545,A 0.000,B 0.000,C 90.000,E1 97.992} C_DIS
LIN {X 0.002,Y -502.740,Z 1600.542,A 0.000,B 0.000,C 90.000,E1 97.530} C_DIS
LIN {X -0.201,Y -503.008,Z 1600.539,A 0.000,B 0.000,C 90.000,E1 97.068} C_DIS
LIN {X 0.102,Y -502.271,Z 1600.536,A 0.000,B 0.000,C 90.000,E1 96.549} C_DIS
LIN {X -0.092,Y -500.407,Z 1600.534,A 0.000,B 0.000,C 90.000,E1 96.087} C_DIS
LIN {X 0.206,Y -497.230,Z 1600.531,A 0.000,B 0.000,C 90.000,E1 95.568} C_DIS
LIN {X 0.160,Y -484.023,Z 1600.520,A 0.000,B 0.000,C 90.000,E1 93.612} C_DIS
LIN {X 0.136,Y -474.060,Z 1600.512,A 0.000,B 0.000,C 90.000,E1 92.121} C_DIS
LIN {X 0.143,Y -465.404,Z 1600.505,A 0.000,B 0.000,C 90.000,E1 90.859} C_DIS
LIN {X -0.202,Y -454.574,Z 1600.496,A 0.000,B 0.000,C 90.000,E1 89.370} C_DIS
LIN {X -0.010,Y -445.128,Z 1600.489,A 0.000,B 0.000,C 90.000,E1 88.051} C_DIS
LIN {X 0.039,Y -435.261,Z 1600.482,A 0.000,B 0.000,C 90.000,E1 86.731} C_DIS
LIN {X -0.198,Y -421.112,Z 1600.471,A 0.000,B 0.000,C 90.000,E1 84.894} C_DIS
LIN {X 0.080,Y -399.971,Z 1600.455,A 0.000,B 0.000,C 90.000,E1 81.837} C_DIS
LIN {X -0.142,Y -380.445,Z 1600.437,A 0.000,B 0.000,C 90.000,E1 78.757} C_DIS
LIN {X -0.008,Y -363.743,Z 1600.421,A 0.000,B 0.000,C 90.000,E1 75.825} C_DIS
LIN {X -0.012,Y -352.426,Z 1600.410,A 0.000,B 0.000,C 90.000,E1 73.740} C_DIS
LIN {X -0.133,Y -339.886,Z 1600.396,A 0.000,B 0.000,C 90.000,E1 71.329} C_DIS
LIN {X -0.072,Y -324.820,Z 1600.379,A 0.000,B 0.000,C 90.000,E1 68.209} C_DIS
LIN {X -0.153,Y -312.148,Z 1600.363,A 0.000,B 0.000,C 90.000,E1 65.357} C_DIS
LIN {X -0.088,Y -301.709,Z 1600.349,A 0.000,B 0.000,C 90.000,E1 62.743} C_DIS
LIN {X 0.132,Y -293.839,Z 1600.337,A 0.000,B 0.000,C 90.000,E1 60.717} C_DIS
LIN {X -0.041,Y -286.987,Z 1600.328,A 0.000,B 0.000,C 90.000,E1 59.076} C_DIS
LIN {X -0.017,Y -279.794,Z 1600.319,A 0.000,B 0.000,C 90.000,E1 57.375} C_DIS
LIN {X -0.015,Y -270.848,Z 1600.307,A 0.000,B 0.000,C 90.000,E1 55.308} C_DIS
LIN {X -0.027,Y -257.585,Z 1600.290,A 0.000,B 0.000,C 90.000,E1 52.145} C_DIS
LIN {X -0.009,Y -245.349,Z 1600.272,A 0.000,B 0.000,C 90.000,E1 48.895} C_DIS
LIN {X 0.002,Y -234.323,Z 1600.253,A 0.000,B 0.000,C 90.000,E1 45.567} C_DIS
LIN {X 0.033,Y -224.334,Z 1600.234,A 0.000,B 0.000,C 90.000,E1 42.162} C_DIS
LIN {X -0.068,Y -216.240,Z 1600.217,A 0.000,B 0.000,C 90.000,E1 39.116} C_DIS
LIN {X 0.034,Y -208.867,Z 1600.200,A 0.000,B 0.000,C 90.000,E1 35.964} C_DIS
LIN {X -0.004,Y -202.267,Z 1600.182,A 0.000,B 0.000,C 90.000,E1 32.801} C_DIS
LIN {X -0.028,Y -196.452,Z 1600.164,A 0.000,B 0.000,C 90.000,E1 29.589} C_DIS
LIN {X 0.038,Y -191.393,Z 1600.146,A 0.000,B 0.000,C 90.000,E1 26.309} C_DIS
LIN {X -0.006,Y -187.026,Z 1600.128,A 0.000,B 0.000,C 90.000,E1 23.025} C_DIS
LIN {X 0.020,Y -182.429,Z 1600.105,A 0.000,B 0.000,C 90.000,E1 18.852} C_DIS
LIN {X -0.035,Y -178.584,Z 1600.081,A 0.000,B 0.000,C 90.000,E1 14.662} C_DIS
LIN {X -0.007,Y -175.030,Z 1600.053,A 0.000,B 0.000,C 90.000,E1 9.557} C_DIS
LIN {X 0.019,Y -172.405,Z 1600.020,A 0.000,B 0.000,C 90.000,E1 3.555} C_DIS
LIN {X 0.050,Y -173.360,Z 1599.926,A 0.000,B 0.000,C 90.000,E1 346.589} C_DIS
LIN {X 0.040,Y -175.938,Z 1599.902,A 0.000,B 0.000,C 90.000,E1 342.308} C_DIS
LIN {X 0.038,Y -178.990,Z 1599.883,A 0.000,B 0.000,C 90.000,E1 338.901} C_DIS
LIN {X -0.023,Y -182.828,Z 1599.864,A 0.000,B 0.000,C 90.000,E1 335.537} C_DIS
LIN {X 0.077,Y -187.402,Z 1599.845,A 0.000,B 0.000,C 90.000,E1 332.153} C_DIS
LIN {X -0.031,Y -192.744,Z 1599.827,A 0.000,B 0.000,C 90.000,E1 328.869} C_DIS
LIN {X -0.041,Y -198.870,Z 1599.809,A 0.000,B 0.000,C 90.000,E1 325.595} C_DIS
LIN {X -0.001,Y -205.751,Z 1599.791,A 0.000,B 0.000,C 90.000,E1 322.351} C_DIS
LIN {X -0.021,Y -213.536,Z 1599.773,A 0.000,B 0.000,C 90.000,E1 319.175} C_DIS
LIN {X -0.024,Y -222.238,Z 1599.756,A 0.000,B 0.000,C 90.000,E1 316.053} C_DIS
LIN {X 0.033,Y -231.870,Z 1599.739,A 0.000,B 0.000,C 90.000,E1 312.975} C_DIS
LIN {X 0.081,Y -241.237,Z 1599.724,A 0.000,B 0.000,C 90.000,E1 310.334} C_DIS
LIN {X -0.013,Y -248.872,Z 1599.714,A 0.000,B 0.000,C 90.000,E1 308.508} C_DIS
LIN {X 0.102,Y -257.510,Z 1599.704,A 0.000,B 0.000,C 90.000,E1 306.664} C_DIS
LIN {X -0.005,Y -267.213,Z 1599.694,A 0.000,B 0.000,C 90.000,E1 304.898} C_DIS
LIN {X -0.078,Y -282.330,Z 1599.680,A 0.000,B 0.000,C 90.000,E1 302.467} C_DIS
LIN {X -0.019,Y -303.902,Z 1599.663,A 0.000,B 0.000,C 90.000,E1 299.411} C_DIS
LIN {X -0.002,Y -316.394,Z 1599.654,A 0.000,B 0.000,C 90.000,E1 297.769} C_DIS
LIN {X 0.054,Y -328.760,Z 1599.645,A 0.000,B 0.000,C 90.000,E1 296.155} C_DIS
LIN {X 0.029,Y -340.950,Z 1599.637,A 0.000,B 0.000,C 90.000,E1 294.591} C_DIS
LIN {X -0.012,Y -360.377,Z 1599.623,A 0.000,B 0.000,C 90.000,E1 292.153} C_DIS
LIN {X -0.012,Y -372.651,Z 1599.615,A 0.000,B 0.000,C 90.000,E1 290.663} C_DIS
LIN {X 0.164,Y -379.783,Z 1599.610,A 0.000,B 0.000,C 90.000,E1 289.758} C_DIS
LIN {X 0.046,Y -386.462,Z 1599.605,A 0.000,B 0.000,C 90.000,E1 288.906} C_DIS
LIN {X -0.009,Y -392.667,Z 1599.600,A 0.000,B 0.000,C 90.000,E1 288.055} C_DIS
LIN {X -0.136,Y -398.296,Z 1599.596,A 0.000,B 0.000,C 90.000,E1 287.221} C_DIS
LIN {X -0.091,Y -403.301,Z 1599.591,A 0.000,B 0.000,C 90.000,E1 286.370} C_DIS
LIN {X 0.072,Y -406.135,Z 1599.588,A 0.000,B 0.000,C 90.000,E1 285.788} C_DIS
LIN {X 0.075,Y -409.630,Z 1599.583,A 0.000,B 0.000,C 90.000,E1 284.954} C_DIS
LIN {X -0.004,Y -411.490,Z 1599.580,A 0.000,B 0.000,C 90.000,E1 284.411} C_DIS
LIN {X -0.181,Y -412.952,Z 1599.577,A 0.000,B 0.000,C 90.000,E1 283.883} C_DIS
LIN {X 0.057,Y -413.921,Z 1599.574,A 0.000,B 0.000,C 90.000,E1 283.300} C_DIS
LIN {X -0.097,Y -414.522,Z 1599.571,A 0.000,B 0.000,C 90.000,E1 282.771} C_DIS
LIN {X 0.160,Y -414.599,Z 1599.568,A 0.000,B 0.000,C 90.000,E1 282.187} C_DIS
LIN {X 0.015,Y -414.201,Z 1599.565,A 0.000,B 0.000,C 90.000,E1 281.658} C_DIS
LIN {X -0.129,Y -413.299,Z 1599.562,A 0.000,B 0.000,C 90.000,E1 281.130} C_DIS
LIN {X 0.129,Y -411.825,Z 1599.559,A 0.000,B 0.000,C 90.000,E1 280.546} C_DIS
LIN {X -0.027,Y -409.703,Z 1599.556,A 0.000,B 0.000,C 90.000,E1 280.018} C_DIS
LIN {X 0.144,Y -406.891,Z 1599.553,A 0.000,B 0.000,C 90.000,E1 279.443} C_DIS
LIN {X -0.041,Y -403.406,Z 1599.550,A 0.000,B 0.000,C 90.000,E1 278.916} C_DIS
LIN {X 0.093,Y -399.191,Z 1599.546,A 0.000,B 0.000,C 90.000,E1 278.341} C_DIS
LIN {X -0.134,Y -394.359,Z 1599.543,A 0.000,B 0.000,C 90.000,E1 277.814} C_DIS
LIN {X -0.049,Y -388.846,Z 1599.540,A 0.000,B 0.000,C 90.000,E1 277.239} C_DIS
LIN {X -0.097,Y -383.066,Z 1599.537,A 0.000,B 0.000,C 90.000,E1 276.720} C_DIS
LIN {X 0.108,Y -377.061,Z 1599.535,A 0.000,B 0.000,C 90.000,E1 276.201} C_DIS
LIN {X -0.174,Y -370.907,Z 1599.532,A 0.000,B 0.000,C 90.000,E1 275.796} C_DIS
LIN {X 0.064,Y -361.489,Z 1599.529,A 0.000,B 0.000,C 90.000,E1 275.163} C_DIS
LIN {X -0.017,Y -351.775,Z 1599.526,A 0.000,B 0.000,C 90.000,E1 274.645} C_DIS
LIN {X -0.096,Y -342.025,Z 1599.523,A 0.000,B 0.000,C 90.000,E1 274.188} C_DIS
LIN {X -0.006,Y -329.067,Z 1599.520,A 0.000,B 0.000,C 90.000,E1 273.612} C_DIS
LIN {X 0.118,Y -319.159,Z 1599.518,A 0.000,B 0.000,C 90.000,E1 273.212} C_DIS
LIN {X -0.136,Y -309.000,Z 1599.516,A 0.000,B 0.000,C 90.000,E1 272.922} C_DIS
LIN {X 0.122,Y -298.357,Z 1599.514,A 0.000,B 0.000,C 90.000,E1 272.579} C_DIS
LIN {X -0.130,Y -291.037,Z 1599.514,A 0.000,B 0.000,C 90.000,E1 272.465} C_DIS
LIN {X 0.006,Y -282.459,Z 1599.513,A 0.000,B 0.000,C 90.000,E1 272.293} C_DIS
LIN {X 0.095,Y -258.942,Z 1599.511,A 0.000,B 0.000,C 90.000,E1 272.007} C_DIS
LIN {X 0.068,Y -242.710,Z 1599.511,A 0.000,B 0.000,C 90.000,E1 271.892} C_DIS
LIN {X 0.074,Y -227.736,Z 1599.510,A 0.000,B 0.000,C 90.000,E1 271.835} C_DIS
LIN {X 0.026,Y -181.288,Z 1599.510,A 0.000,B 0.000,C 90.000,E1 271.835} C_DIS
LIN {X 0.006,Y -181.574,Z 1599.501,A 0.000,B 0.000,C 90.000,E1 270.115} C_DIS
LIN {X -0.006,Y -180.875,Z 1599.473,A 0.000,B 0.000,C 90.000,E1 265.065} C_DIS
LIN {X 0.051,Y -178.992,Z 1599.444,A 0.000,B 0.000,C 90.000,E1 259.982} C_DIS
LIN {X 0.062,Y -177.981,Z 1599.435,A 0.000,B 0.000,C 90.000,E1 258.285} C_DIS
LIN {X 0.031,Y -175.624,Z 1599.411,A 0.000,B 0.000,C 90.000,E1 254.047} C_DIS
LIN {X 0.091,Y -172.345,Z 1599.388,A 0.000,B 0.000,C 90.000,E1 249.752} C_DIS
LIN {X 0.044,Y -171.124,Z 1599.378,A 0.000,B 0.000,C 90.000,E1 248.050} C_DIS
LIN {X -0.070,Y -167.432,Z 1599.354,A 0.000,B 0.000,C 90.000,E1 243.768} C_DIS
LIN {X 0.013,Y -166.828,Z 1599.349,A 0.000,B 0.000,C 90.000,E1 242.871} C_DIS
LIN {X -0.070,Y -162.811,Z 1599.325,A 0.000,B 0.000,C 90.000,E1 238.535} C_DIS
LIN {X -0.006,Y -161.498,Z 1599.315,A 0.000,B 0.000,C 90.000,E1 236.755} C_DIS
LIN {X -0.053,Y -157.495,Z 1599.291,A 0.000,B 0.000,C 90.000,E1 232.351} C_DIS
LIN {X -0.018,Y -155.514,Z 1599.276,A 0.000,B 0.000,C 90.000,E1 229.666} C_DIS
LIN {X 0.032,Y -151.814,Z 1599.251,A 0.000,B 0.000,C 90.000,E1 225.162} C_DIS
LIN {X 0.044,Y -150.027,Z 1599.236,A 0.000,B 0.000,C 90.000,E1 222.447} C_DIS
LIN {X -0.041,Y -146.848,Z 1599.211,A 0.000,B 0.000,C 90.000,E1 217.935} C_DIS
LIN {X -0.023,Y -145.431,Z 1599.195,A 0.000,B 0.000,C 90.000,E1 215.185} C_DIS
LIN {X -0.028,Y -142.854,Z 1599.170,A 0.000,B 0.000,C 90.000,E1 210.590} C_DIS
LIN {X 0.025,Y -141.469,Z 1599.149,A 0.000,B 0.000,C 90.000,E1 206.873} C_DIS
LIN {X 0.016,Y -139.378,Z 1599.113,A 0.000,B 0.000,C 90.000,E1 200.375} C_DIS
LIN {X 0.006,Y -138.830,Z 1599.098,A 0.000,B 0.000,C 90.000,E1 197.583} C_DIS
LIN {X -0.066,Y -138.354,Z 1599.056,A 0.000,B 0.000,C 90.000,E1 190.141} C_DIS
LIN {X 0.068,Y -139.528,Z 1599.004,A 0.000,B 0.000,C 90.000,E1 180.745} C_DIS
LIN {X 0.021,Y -141.201,Z 1598.973,A 0.000,B 0.000,C 90.000,E1 175.179} C_DIS
LIN {X -0.019,Y -142.577,Z 1598.958,A 0.000,B 0.000,C 90.000,E1 172.413} C_DIS
LIN {X 0.076,Y -144.869,Z 1598.932,A 0.000,B 0.000,C 90.000,E1 167.757} C_DIS
LIN {X 0.031,Y -147.495,Z 1598.912,A 0.000,B 0.000,C 90.000,E1 164.102} C_DIS
LIN {X -0.036,Y -150.084,Z 1598.891,A 0.000,B 0.000,C 90.000,E1 160.477} C_DIS
LIN {X -0.022,Y -153.437,Z 1598.871,A 0.000,B 0.000,C 90.000,E1 156.847} C_DIS
LIN {X -0.028,Y -157.799,Z 1598.846,A 0.000,B 0.000,C 90.000,E1 152.359} C_DIS
LIN {X 0.005,Y -162.080,Z 1598.827,A 0.000,B 0.000,C 90.000,E1 148.791} C_DIS
LIN {X 0.030,Y -166.280,Z 1598.807,A 0.000,B 0.000,C 90.000,E1 145.261} C_DIS
LIN {X 0.027,Y -171.296,Z 1598.788,A 0.000,B 0.000,C 90.000,E1 141.778} C_DIS
LIN {X 0.062,Y -176.191,Z 1598.769,A 0.000,B 0.000,C 90.000,E1 138.324} C_DIS
LIN {X -0.072,Y -180.466,Z 1598.754,A 0.000,B 0.000,C 90.000,E1 135.810} C_DIS
LIN {X -0.097,Y -185.871,Z 1598.736,A 0.000,B 0.000,C 90.000,E1 132.447} C_DIS
LIN {X -0.045,Y -190.496,Z 1598.722,A 0.000,B 0.000,C 90.000,E1 129.930} C_DIS
LIN {X -0.024,Y -196.247,Z 1598.703,A 0.000,B 0.000,C 90.000,E1 126.629} C_DIS
LIN {X -0.066,Y -201.053,Z 1598.690,A 0.000,B 0.000,C 90.000,E1 124.199} C_DIS
LIN {X 0.035,Y -204.927,Z 1598.678,A 0.000,B 0.000,C 90.000,E1 122.005} C_DIS
LIN {X 0.018,Y -322.612,Z 1598.678,A 0.000,B 0.000,C 90.000,E1 122.005} C_DIS
LIN {X -0.098,Y -324.219,Z 1598.678,A 0.000,B 0.000,C 90.000,E1 122.005} C_DIS
LIN {X 0.071,Y -329.415,Z 1598.677,A 0.000,B 0.000,C 90.000,E1 121.750} C_DIS
LIN {X 0.163,Y -332.544,Z 1598.675,A 0.000,B 0.000,C 90.000,E1 121.465} C_DIS
LIN {X -0.022,Y -336.209,Z 1598.672,A 0.000,B 0.000,C 90.000,E1 121.003} C_DIS
LIN {X 0.106,Y -337.832,Z 1598.671,A 0.000,B 0.000,C 90.000,E1 120.669} C_DIS
LIN {X 0.109,Y -350.971,Z 1598.653,A 0.000,B 0.000,C 90.000,E1 117.590} C_DIS
LIN {X -0.014,Y -364.259,Z 1598.638,A 0.000,B 0.000,C 90.000,E1 114.899} C_DIS
LIN {X -0.082,Y -379.100,Z 1598.624,A 0.000,B 0.000,C 90.000,E1 112.259} C_DIS
LIN {X 0.028,Y -393.706,Z 1598.611,A 0.000,B 0.000,C 90.000,E1 109.939} C_DIS
LIN {X 0.003,Y -409.744,Z 1598.598,A 0.000,B 0.000,C 90.000,E1 107.692} C_DIS
LIN {X 0.122,Y -427.325,Z 1598.586,A 0.000,B 0.000,C 90.000,E1 105.481} C_DIS
LIN {X 0.077,Y -446.524,Z 1598.574,A 0.000,B 0.000,C 90.000,E1 103.355} C_DIS
LIN {X 0.081,Y -466.615,Z 1598.563,A 0.000,B 0.000,C 90.000,E1 101.366} C_DIS
LIN {X 0.063,Y -489.866,Z 1598.552,A 0.000,B 0.000,C 90.000,E1 99.321} C_DIS
LIN {X -0.148,Y -495.105,Z 1598.549,A 0.000,B 0.000,C 90.000,E1 98.916} C_DIS
LIN {X 0.040,Y -497.280,Z 1598.548,A 0.000,B 0.000,C 90.000,E1 98.681} C_DIS
LIN {X 0.155,Y -498.933,Z 1598.547,A 0.000,B 0.000,C 90.000,E1 98.454} C_DIS
LIN {X 0.077,Y -500.374,Z 1598.546,A 0.000,B 0.000,C 90.000,E1 98.219} C_DIS
LIN {X -0.073,Y -501.439,Z 1598.544,A 0.000,B 0.000,C 90.000,E1 97.992} C_DIS
LIN {X 0.216,Y -502.663,Z 1598.542,A 0.000,B 0.000,C 90.000,E1 97.473} C_DIS
LIN {X 0.075,Y -502.848,Z 1598.539,A 0.000,B 0.000,C 90.000,E1 97.004} C_DIS
LIN {X -0.125,Y -502.024,Z 1598.536,A 0.000,B 0.000,C 90.000,E1 96.543} C_DIS
LIN {X 0.121,Y -500.053,Z 1598.534,A 0.000,B 0.000,C 90.000,E1 96.030} C_DIS
LIN {X -0.164,Y -495.126,Z 1598.530,A 0.000,B 0.000,C 90.000,E1 95.334} C_DIS
LIN {X -0.124,Y -483.643,Z 1598.520,A 0.000,B 0.000,C 90.000,E1 93.612} C_DIS
LIN {X -0.150,Y -473.664,Z 1598.512,A 0.000,B 0.000,C 90.000,E1 92.121} C_DIS
LIN {X -0.143,Y -465.010,Z 1598.505,A 0.000,B 0.000,C 90.000,E1 90.859} C_DIS
LIN {X -0.033,Y -454.177,Z 1598.496,A 0.000,B 0.000,C 90.000,E1 89.312} C_DIS
LIN {X 0.149,Y -444.714,Z 1598.489,A 0.000,B 0.000,C 90.000,E1 87.993} C_DIS
LIN {X 0.189,Y -434.834,Z 1598.482,A 0.000,B 0.000,C 90.000,E1 86.674} C_DIS
LIN {X -0.062,Y -420.678,Z 1598.471,A 0.000,B 0.000,C 90.000,E1 84.837} C_DIS
LIN {X 0.160,Y -401.427,Z 1598.456,A 0.000,B 0.000,C 90.000,E1 82.064} C_DIS
LIN {X -0.087,Y -381.783,Z 1598.439,A 0.000,B 0.000,C 90.000,E1 78.993} C_DIS
LIN {X 0.100,Y -366.665,Z 1598.424,A 0.000,B 0.000,C 90.000,E1 76.353} C_DIS
LIN {X 0.107,Y -353.700,Z 1598.411,A 0.000,B 0.000,C 90.000,E1 73.976} C_DIS
LIN {X -0.093,Y -341.103,Z 1598.398,A 0.000,B 0.000,C 90.000,E1 71.583} C_DIS
LIN {X 0.021,Y -327.436,Z 1598.382,A 0.000,B 0.000,C 90.000,E1 68.773} C_DIS
LIN {X -0.012,Y -311.794,Z 1598.363,A 0.000,B 0.000,C 90.000,E1 65.281} C_DIS
LIN {X 0.047,Y -301.321,Z 1598.348,A 0.000,B 0.000,C 90.000,E1 62.666} C_DIS
LIN {X 0.115,Y -293.413,Z 1598.337,A 0.000,B 0.000,C 90.000,E1 60.667} C_DIS
LIN {X 0.080,Y -286.524,Z 1598.328,A 0.000,B 0.000,C 90.000,E1 58.997} C_DIS
LIN {X -0.054,Y -279.296,Z 1598.318,A 0.000,B 0.000,C 90.000,E1 57.327} C_DIS
LIN {X -0.065,Y -270.344,Z 1598.307,A 0.000,B 0.000,C 90.000,E1 55.261} C_DIS
LIN {X 0.061,Y -257.180,Z 1598.289,A 0.000,B 0.000,C 90.000,E1 52.065} C_DIS
LIN {X -0.095,Y -245.041,Z 1598.271,A 0.000,B 0.000,C 90.000,E1 48.852} C_DIS
LIN {X 0.067,Y -234.067,Z 1598.253,A 0.000,B 0.000,C 90.000,E1 45.486} C_DIS
LIN {X 0.088,Y -224.120,Z 1598.234,A 0.000,B 0.000,C 90.000,E1 42.081} C_DIS
LIN {X -0.021,Y -216.061,Z 1598.217,A 0.000,B 0.000,C 90.000,E1 39.036} C_DIS
LIN {X 0.072,Y -208.724,Z 1598.199,A 0.000,B 0.000,C 90.000,E1 35.884} C_DIS
LIN {X -0.082,Y -202.166,Z 1598.182,A 0.000,B 0.000,C 90.000,E1 32.752} C_DIS
LIN {X -0.101,Y -196.388,Z 1598.164,A 0.000,B 0.000,C 90.000,E1 29.539} C_DIS
LIN {X 0.056,Y -191.368,Z 1598.146,A 0.000,B 0.000,C 90.000,E1 26.232} C_DIS
LIN {X -0.097,Y -186.046,Z 1598.123,A 0.000,B 0.000,C 90.000,E1 22.153} C_DIS
LIN {X 0.010,Y -181.637,Z 1598.100,A 0.000,B 0.000,C 90.000,E1 17.946} C_DIS
LIN {X 0.052,Y -177.993,Z 1598.076,A 0.000,B 0.000,C 90.000,E1 13.716} C_DIS
LIN {X 0.020,Y -174.699,Z 1598.048,A 0.000,B 0.000,C 90.000,E1 8.624} C_DIS
LIN {X -0.006,Y -172.258,Z 1598.015,A 0.000,B 0.000,C 90.000,E1 2.636} C_DIS
LIN {X 0.017,Y -173.191,Z 1597.930,A 0.000,B 0.000,C 90.000,E1 347.465} C_DIS
LIN {X 0.066,Y -176.174,Z 1597.902,A 0.000,B 0.000,C 90.000,E1 342.308} C_DIS
LIN {X -0.086,Y -180.114,Z 1597.878,A 0.000,B 0.000,C 90.000,E1 338.103} C_DIS
LIN {X -0.049,Y -184.114,Z 1597.859,A 0.000,B 0.000,C 90.000,E1 334.717} C_DIS
LIN {X -0.086,Y -188.868,Z 1597.841,A 0.000,B 0.000,C 90.000,E1 331.385} C_DIS
LIN {X -0.071,Y -194.374,Z 1597.823,A 0.000,B 0.000,C 90.000,E1 328.074} C_DIS
LIN {X 0.066,Y -200.652,Z 1597.804,A 0.000,B 0.000,C 90.000,E1 324.769} C_DIS
LIN {X 0.113,Y -207.704,Z 1597.786,A 0.000,B 0.000,C 90.000,E1 321.537} C_DIS
LIN {X -0.015,Y -215.668,Z 1597.769,A 0.000,B 0.000,C 90.000,E1 318.405} C_DIS
LIN {X -0.123,Y -224.575,Z 1597.752,A 0.000,B 0.000,C 90.000,E1 315.324} C_DIS
LIN {X 0.004,Y -234.423,Z 1597.735,A 0.000,B 0.000,C 90.000,E1 312.243} C_DIS
LIN {X -0.054,Y -242.618,Z 1597.722,A 0.000,B 0.000,C 90.000,E1 310.011} C_DIS
LIN {X -0.090,Y -250.406,Z 1597.712,A 0.000,B 0.000,C 90.000,E1 308.177} C_DIS
LIN {X -0.159,Y -259.208,Z 1597.702,A 0.000,B 0.000,C 90.000,E1 306.377} C_DIS
LIN {X 0.039,Y -271.211,Z 1597.690,A 0.000,B 0.000,C 90.000,E1 304.199} C_DIS
LIN {X -0.096,Y -286.771,Z 1597.677,A 0.000,B 0.000,C 90.000,E1 301.799} C_DIS
LIN {X 0.100,Y -308.759,Z 1597.660,A 0.000,B 0.000,C 90.000,E1 298.743} C_DIS
LIN {X 0.047,Y -321.205,Z 1597.651,A 0.000,B 0.000,C 90.000,E1 297.129} C_DIS
LIN {X 0.040,Y -333.547,Z 1597.642,A 0.000,B 0.000,C 90.000,E1 295.540} C_DIS
LIN {X 0.096,Y -343.216,Z 1597.635,A 0.000,B 0.000,C 90.000,E1 294.283} C_DIS
LIN {X 0.120,Y -362.782,Z 1597.621,A 0.000,B 0.000,C 90.000,E1 291.844} C_DIS
LIN {X 0.035,Y -375.041,Z 1597.613,A 0.000,B 0.000,C 90.000,E1 290.375} C_DIS
LIN {X 0.002,Y -382.061,Z 1597.608,A 0.000,B 0.000,C 90.000,E1 289.504} C_DIS
LIN {X -0.090,Y -388.622,Z 1597.604,A 0.000,B 0.000,C 90.000,E1 288.652} C_DIS
LIN {X 0.118,Y -394.679,Z 1597.599,A 0.000,B 0.000,C 90.000,E1 287.764} C_DIS
LIN {X 0.137,Y -400.141,Z 1597.594,A 0.000,B 0.000,C 90.000,E1 286.913} C_DIS
LIN {X 0.081,Y -404.953,Z 1597.589,A 0.000,B 0.000,C 90.000,E1 286.079} C_DIS
LIN {X -0.133,Y -407.608,Z 1597.586,A 0.000,B 0.000,C 90.000,E1 285.552} C_DIS
LIN {X 0.174,Y -409.852,Z 1597.583,A 0.000,B 0.000,C 90.000,E1 284.954} C_DIS
LIN {X -0.006,Y -411.749,Z 1597.580,A 0.000,B 0.000,C 90.000,E1 284.426} C_DIS
LIN {X -0.078,Y -413.203,Z 1597.577,A 0.000,B 0.000,C 90.000,E1 283.883} C_DIS
LIN {X 0.161,Y -414.246,Z 1597.574,A 0.000,B 0.000,C 90.000,E1 283.300} C_DIS
LIN {X 0.008,Y -414.848,Z 1597.571,A 0.000,B 0.000,C 90.000,E1 282.771} C_DIS
LIN {X -0.138,Y -414.966,Z 1597.568,A 0.000,B 0.000,C 90.000,E1 282.243} C_DIS
LIN {X 0.125,Y -414.637,Z 1597.565,A 0.000,B 0.000,C 90.000,E1 281.658} C_DIS
LIN {X -0.017,Y -413.747,Z 1597.562,A 0.000,B 0.000,C 90.000,E1 281.130} C_DIS
LIN {X -0.163,Y -412.315,Z 1597.559,A 0.000,B 0.000,C 90.000,E1 280.602} C_DIS
LIN {X 0.089,Y -410.219,Z 1597.556,A 0.000,B 0.000,C 90.000,E1 280.018} C_DIS
LIN {X -0.141,Y -407.471,Z 1597.553,A 0.000,B 0.000,C 90.000,E1 279.500} C_DIS
LIN {X 0.079,Y -403.989,Z 1597.550,A 0.000,B 0.000,C 90.000,E1 278.916} C_DIS
LIN {X -0.181,Y -399.820,Z 1597.547,A 0.000,B 0.000,C 90.000,E1 278.398} C_DIS
LIN {X -0.009,Y -394.988,Z 1597.543,A 0.000,B 0.000,C 90.000,E1 277.814} C_DIS
LIN {X 0.078,Y -389.500,Z 1597.540,A 0.000,B 0.000,C 90.000,E1 277.239} C_DIS
LIN {X 0.014,Y -383.683,Z 1597.537,A 0.000,B 0.000,C 90.000,E1 276.720} C_DIS
LIN {X -0.129,Y -377.764,Z 1597.535,A 0.000,B 0.000,C 90.000,E1 276.258} C_DIS
LIN {X -0.036,Y -371.572,Z 1597.532,A 0.000,B 0.000,C 90.000,E1 275.796} C_DIS
LIN {X -0.038,Y -365.383,Z 1597.530,A 0.000,B 0.000,C 90.000,E1 275.391} C_DIS
LIN {X 0.105,Y -358.957,Z 1597.528,A 0.000,B 0.000,C 90.000,E1 274.992} C_DIS
LIN {X -0.171,Y -349.226,Z 1597.525,A 0.000,B 0.000,C 90.000,E1 274.531} C_DIS
LIN {X -0.144,Y -339.388,Z 1597.522,A 0.000,B 0.000,C 90.000,E1 274.069} C_DIS
LIN {X 0.130,Y -329.761,Z 1597.520,A 0.000,B 0.000,C 90.000,E1 273.612} C_DIS
LIN {X -0.070,Y -319.894,Z 1597.518,A 0.000,B 0.000,C 90.000,E1 273.269} C_DIS
LIN {X 0.023,Y -306.334,Z 1597.516,A 0.000,B 0.000,C 90.000,E1 272.808} C_DIS
LIN {X 0.058,Y -295.484,Z 1597.514,A 0.000,B 0.000,C 90.000,E1 272.522} C_DIS
LIN {X -0.140,Y -287.682,Z 1597.513,A 0.000,B 0.000,C 90.000,E1 272.407} C_DIS
LIN {X 0.070,Y -273.831,Z 1597.512,A 0.000,B 0.000,C 90.000,E1 272.178} C_DIS
LIN {X -0.096,Y -260.325,Z 1597.511,A 0.000,B 0.000,C 90.000,E1 272.064} C_DIS
LIN {X -0.110,Y -245.051,Z 1597.511,A 0.000,B 0.000,C 90.000,E1 271.949} C_DIS
LIN {X -0.094,Y -231.015,Z 1597.510,A 0.000,B 0.000,C 90.000,E1 271.892} C_DIS
LIN {X 0.074,Y -181.285,Z 1597.510,A 0.000,B 0.000,C 90.000,E1 271.835} C_DIS
LIN {X 0.054,Y -181.575,Z 1597.501,A 0.000,B 0.000,C 90.000,E1 270.115} C_DIS
LIN {X 0.042,Y -180.878,Z 1597.473,A 0.000,B 0.000,C 90.000,E1 265.065} C_DIS
LIN {X -0.078,Y -178.996,Z 1597.445,A 0.000,B 0.000,C 90.000,E1 260.038} C_DIS
LIN {X 0.016,Y -178.582,Z 1597.440,A 0.000,B 0.000,C 90.000,E1 259.162} C_DIS
LIN {X -0.090,Y -175.636,Z 1597.411,A 0.000,B 0.000,C 90.000,E1 254.102} C_DIS
LIN {X -0.024,Y -172.355,Z 1597.388,A 0.000,B 0.000,C 90.000,E1 249.806} C_DIS
LIN {X -0.069,Y -171.140,Z 1597.378,A 0.000,B 0.000,C 90.000,E1 248.103} C_DIS
LIN {X -0.024,Y -167.444,Z 1597.354,A 0.000,B 0.000,C 90.000,E1 243.768} C_DIS
LIN {X 0.058,Y -166.840,Z 1597.349,A 0.000,B 0.000,C 90.000,E1 242.871} C_DIS
LIN {X -0.025,Y -162.823,Z 1597.325,A 0.000,B 0.000,C 90.000,E1 238.535} C_DIS
LIN {X 0.039,Y -161.509,Z 1597.315,A 0.000,B 0.000,C 90.000,E1 236.755} C_DIS
LIN {X -0.008,Y -157.507,Z 1597.291,A 0.000,B 0.000,C 90.000,E1 232.351} C_DIS
LIN {X 0.026,Y -155.529,Z 1597.276,A 0.000,B 0.000,C 90.000,E1 229.666} C_DIS
LIN {X 0.075,Y -151.826,Z 1597.251,A 0.000,B 0.000,C 90.000,E1 225.162} C_DIS
LIN {X 0.087,Y -150.040,Z 1597.236,A 0.000,B 0.000,C 90.000,E1 222.447} C_DIS
LIN {X 0.001,Y -146.857,Z 1597.211,A 0.000,B 0.000,C 90.000,E1 217.935} C_DIS
LIN {X 0.019,Y -145.441,Z 1597.196,A 0.000,B 0.000,C 90.000,E1 215.185} C_DIS
LIN {X 0.014,Y -142.862,Z 1597.170,A 0.000,B 0.000,C 90.000,E1 210.590} C_DIS
LIN {X 0.066,Y -141.478,Z 1597.149,A 0.000,B 0.000,C 90.000,E1 206.873} C_DIS
LIN {X -0.074,Y -139.380,Z 1597.113,A 0.000,B 0.000,C 90.000,E1 200.429} C_DIS
LIN {X 0.047,Y -138.834,Z 1597.098,A 0.000,B 0.000,C 90.000,E1 197.583} C_DIS
LIN {X -0.025,Y -138.354,Z 1597.056,A 0.000,B 0.000,C 90.000,E1 190.141} C_DIS
LIN {X -0.030,Y -139.524,Z 1597.004,A 0.000,B 0.000,C 90.000,E1 180.802} C_DIS
LIN {X 0.063,Y -141.193,Z 1596.973,A 0.000,B 0.000,C 90.000,E1 175.179} C_DIS
LIN {X 0.022,Y -142.570,Z 1596.958,A 0.000,B 0.000,C 90.000,E1 172.413} C_DIS
LIN {X -0.023,Y -144.858,Z 1596.932,A 0.000,B 0.000,C 90.000,E1 167.813} C_DIS
LIN {X -0.068,Y -147.484,Z 1596.912,A 0.000,B 0.000,C 90.000,E1 164.157} C_DIS
LIN {X -0.042,Y -150.071,Z 1596.892,A 0.000,B 0.000,C 90.000,E1 160.496} C_DIS
LIN {X -0.039,Y -153.420,Z 1596.871,A 0.000,B 0.000,C 90.000,E1 156.869} C_DIS
LIN {X 0.010,Y -156.840,Z 1596.851,A 0.000,B 0.000,C 90.000,E1 153.256} C_DIS
LIN {X 0.081,Y -160.920,Z 1596.832,A 0.000,B 0.000,C 90.000,E1 149.665} C_DIS
LIN {X 0.026,Y -163.045,Z 1596.822,A 0.000,B 0.000,C 90.000,E1 147.916} C_DIS
LIN {X 0.030,Y -167.437,Z 1596.802,A 0.000,B 0.000,C 90.000,E1 144.402} C_DIS
LIN {X -0.060,Y -171.275,Z 1596.788,A 0.000,B 0.000,C 90.000,E1 141.823} C_DIS
LIN {X -0.021,Y -176.167,Z 1596.769,A 0.000,B 0.000,C 90.000,E1 138.366} C_DIS
LIN {X -0.024,Y -180.440,Z 1596.755,A 0.000,B 0.000,C 90.000,E1 135.810} C_DIS
LIN {X -0.048,Y -185.845,Z 1596.736,A 0.000,B 0.000,C 90.000,E1 132.447} C_DIS
LIN {X 0.005,Y -190.467,Z 1596.722,A 0.000,B 0.000,C 90.000,E1 129.930} C_DIS
LIN {X -0.090,Y -196.219,Z 1596.703,A 0.000,B 0.000,C 90.000,E1 126.664} C_DIS
LIN {X -0.015,Y -201.029,Z 1596.690,A 0.000,B 0.000,C 90.000,E1 124.199} C_DIS
LIN {X -0.030,Y -204.869,Z 1596.678,A 0.000,B 0.000,C 90.000,E1 122.054} C_DIS
LIN {X 0.184,Y -323.133,Z 1596.678,A 0.000,B 0.000,C 90.000,E1 122.005} C_DIS
LIN {X -0.125,Y -329.553,Z 1596.677,A 0.000,B 0.000,C 90.000,E1 121.799} C_DIS
LIN {X -0.026,Y -332.564,Z 1596.675,A 0.000,B 0.000,C 90.000,E1 121.514} C_DIS
LIN {X 0.001,Y -336.233,Z 1596.672,A 0.000,B 0.000,C 90.000,E1 121.003} C_DIS
LIN {X 0.128,Y -337.814,Z 1596.671,A 0.000,B 0.000,C 90.000,E1 120.669} C_DIS
LIN {X 0.132,Y -350.932,Z 1596.653,A 0.000,B 0.000,C 90.000,E1 117.590} C_DIS
LIN {X 0.009,Y -364.217,Z 1596.638,A 0.000,B 0.000,C 90.000,E1 114.899} C_DIS
LIN {X -0.060,Y -379.056,Z 1596.624,A 0.000,B 0.000,C 90.000,E1 112.259} C_DIS
LIN {X 0.049,Y -393.659,Z 1596.611,A 0.000,B 0.000,C 90.000,E1 109.939} C_DIS
LIN {X 0.025,Y -409.695,Z 1596.598,A 0.000,B 0.000,C 90.000,E1 107.692} C_DIS
LIN {X 0.144,Y -427.274,Z 1596.586,A 0.000,B 0.000,C 90.000,E1 105.481} C_DIS
LIN {X 0.097,Y -446.472,Z 1596.574,A 0.000,B 0.000,C 90.000,E1 103.355} C_DIS
LIN {X 0.100,Y -466.561,Z 1596.563,A 0.000,B 0.000,C 90.000,E1 101.366} C_DIS
LIN {X 0.080,Y -489.811,Z 1596.552,A 0.000,B 0.000,C 90.000,E1 99.321} C_DIS
LIN {X -0.131,Y -495.046,Z 1596.549,A 0.000,B 0.000,C 90.000,E1 98.916} C_DIS
LIN {X 0.055,Y -497.200,Z 1596.548,A 0.000,B 0.000,C 90.000,E1 98.681} C_DIS
LIN {X 0.166,Y -498.840,Z 1596.547,A 0.000,B 0.000,C 90.000,E1 98.454} C_DIS
LIN {X 0.089,Y -500.267,Z 1596.546,A 0.000,B 0.000,C 90.000,E1 98.219} C_DIS
LIN {X -0.061,Y -501.324,Z 1596.544,A 0.000,B 0.000,C 90.000,E1 97.992} C_DIS
LIN {X -0.271,Y -502.531,Z 1596.542,A 0.000,B 0.000,C 90.000,E1 97.530} C_DIS
LIN {X 0.086,Y -502.702,Z 1596.539,A 0.000,B 0.000,C 90.000,E1 97.004} C_DIS
LIN {X -0.115,Y -501.864,Z 1596.536,A 0.000,B 0.000,C 90.000,E1 96.543} C_DIS
LIN {X 0.130,Y -499.873,Z 1596.534,A 0.000,B 0.000,C 90.000,E1 96.030} C_DIS
LIN {X 0.061,Y -491.654,Z 1596.527,A 0.000,B 0.000,C 90.000,E1 94.821} C_DIS
LIN {X 0.065,Y -480.185,Z 1596.517,A 0.000,B 0.000,C 90.000,E1 93.094} C_DIS
LIN {X -0.028,Y -470.085,Z 1596.509,A 0.000,B 0.000,C 90.000,E1 91.604} C_DIS
LIN {X -0.088,Y -461.291,Z 1596.502,A 0.000,B 0.000,C 90.000,E1 90.344} C_DIS
LIN {X 0.191,Y -452.185,Z 1596.495,A 0.000,B 0.000,C 90.000,E1 89.026} C_DIS
LIN {X -0.108,Y -442.630,Z 1596.488,A 0.000,B 0.000,C 90.000,E1 87.764} C_DIS
LIN {X 0.058,Y -430.658,Z 1596.479,A 0.000,B 0.000,C 90.000,E1 86.159} C_DIS
LIN {X 0.059,Y -410.698,Z 1596.464,A 0.000,B 0.000,C 90.000,E1 83.457} C_DIS
LIN {X 0.104,Y -390.418,Z 1596.447,A 0.000,B 0.000,C 90.000,E1 80.387} C_DIS
LIN {X 0.088,Y -373.178,Z 1596.431,A 0.000,B 0.000,C 90.000,E1 77.521} C_DIS
LIN {X 0.128,Y -358.419,Z 1596.416,A 0.000,B 0.000,C 90.000,E1 74.866} C_DIS
LIN {X -0.059,Y -345.675,Z 1596.403,A 0.000,B 0.000,C 90.000,E1 72.489} C_DIS
LIN {X 0.067,Y -331.797,Z 1596.387,A 0.000,B 0.000,C 90.000,E1 69.699} C_DIS
LIN {X 0.107,Y -317.189,Z 1596.370,A 0.000,B 0.000,C 90.000,E1 66.538} C_DIS
LIN {X -0.013,Y -302.420,Z 1596.350,A 0.000,B 0.000,C 90.000,E1 62.999} C_DIS
LIN {X 0.076,Y -294.536,Z 1596.339,A 0.000,B 0.000,C 90.000,E1 61.001} C_DIS
LIN {X 0.043,Y -286.272,Z 1596.328,A 0.000,B 0.000,C 90.000,E1 58.997} C_DIS
LIN {X -0.094,Y -279.019,Z 1596.318,A 0.000,B 0.000,C 90.000,E1 57.327} C_DIS
LIN {X -0.109,Y -270.089,Z 1596.307,A 0.000,B 0.000,C 90.000,E1 55.261} C_DIS
LIN {X 0.013,Y -257.000,Z 1596.289,A 0.000,B 0.000,C 90.000,E1 52.065} C_DIS
LIN {X -0.146,Y -244.917,Z 1596.271,A 0.000,B 0.000,C 90.000,E1 48.852} C_DIS
LIN {X 0.016,Y -233.979,Z 1596.253,A 0.000,B 0.000,C 90.000,E1 45.486} C_DIS
LIN {X 0.043,Y -224.069,Z 1596.234,A 0.000,B 0.000,C 90.000,E1 42.081} C_DIS
LIN {X -0.066,Y -216.024,Z 1596.217,A 0.000,B 0.000,C 90.000,E1 39.036} C_DIS
LIN {X 0.028,Y -208.709,Z 1596.199,A 0.000,B 0.000,C 90.000,E1 35.884} C_DIS
LIN {X 0.045,Y -202.185,Z 1596.182,A 0.000,B 0.000,C 90.000,E1 32.704} C_DIS
LIN {X 0.029,Y -196.422,Z 1596.164,A 0.000,B 0.000,C 90.000,E1 29.489} C_DIS
LIN {X 0.017,Y -191.431,Z 1596.146,A 0.000,B 0.000,C 90.000,E1 26.232} C_DIS
LIN {X 0.039,Y -186.140,Z 1596.123,A 0.000,B 0.000,C 90.000,E1 22.099} C_DIS
LIN {X -0.023,Y -181.745,Z 1596.100,A 0.000,B 0.000,C 90.000,E1 17.946} C_DIS
LIN {X 0.025,Y -178.118,Z 1596.076,A 0.000,B 0.000,C 90.000,E1 13.716} C_DIS
LIN {X -0.002,Y -174.869,Z 1596.048,A 0.000,B 0.000,C 90.000,E1 8.624} C_DIS
LIN {X -0.030,Y -172.716,Z 1596.019,A 0.000,B 0.000,C 90.000,E1 3.498} C_DIS
LIN {X 0.035,Y -173.422,Z 1595.930,A 0.000,B 0.000,C 90.000,E1 347.465} C_DIS
LIN {X -0.074,Y -176.429,Z 1595.902,A 0.000,B 0.000,C 90.000,E1 342.362} C_DIS
LIN {X -0.051,Y -180.344,Z 1595.878,A 0.000,B 0.000,C 90.000,E1 338.103} C_DIS
LIN {X -0.007,Y -184.327,Z 1595.859,A 0.000,B 0.000,C 90.000,E1 334.717} C_DIS
LIN {X -0.039,Y -189.068,Z 1595.841,A 0.000,B 0.000,C 90.000,E1 331.385} C_DIS
LIN {X -0.017,Y -194.534,Z 1595.823,A 0.000,B 0.000,C 90.000,E1 328.074} C_DIS
LIN {X -0.038,Y -200.791,Z 1595.804,A 0.000,B 0.000,C 90.000,E1 324.815} C_DIS
LIN {X -0.113,Y -207.800,Z 1595.787,A 0.000,B 0.000,C 90.000,E1 321.618} C_DIS
LIN {X 0.056,Y -215.722,Z 1595.769,A 0.000,B 0.000,C 90.000,E1 318.405} C_DIS
LIN {X -0.049,Y -224.590,Z 1595.752,A 0.000,B 0.000,C 90.000,E1 315.324} C_DIS
LIN {X -0.092,Y -234.385,Z 1595.735,A 0.000,B 0.000,C 90.000,E1 312.285} C_DIS
LIN {X 0.026,Y -242.531,Z 1595.722,A 0.000,B 0.000,C 90.000,E1 310.011} C_DIS
LIN {X -0.008,Y -250.293,Z 1595.712,A 0.000,B 0.000,C 90.000,E1 308.177} C_DIS
LIN {X -0.078,Y -259.094,Z 1595.702,A 0.000,B 0.000,C 90.000,E1 306.377} C_DIS
LIN {X 0.123,Y -271.055,Z 1595.690,A 0.000,B 0.000,C 90.000,E1 304.199} C_DIS
LIN {X -0.012,Y -286.606,Z 1595.677,A 0.000,B 0.000,C 90.000,E1 301.799} C_DIS
LIN {X 0.036,Y -308.620,Z 1595.660,A 0.000,B 0.000,C 90.000,E1 298.771} C_DIS
LIN {X 0.134,Y -321.049,Z 1595.651,A 0.000,B 0.000,C 90.000,E1 297.129} C_DIS
LIN {X 0.127,Y -333.410,Z 1595.642,A 0.000,B 0.000,C 90.000,E1 295.540} C_DIS
LIN {X 0.012,Y -345.517,Z 1595.633,A 0.000,B 0.000,C 90.000,E1 294.003} C_DIS
LIN {X -0.063,Y -365.165,Z 1595.620,A 0.000,B 0.000,C 90.000,E1 291.589} C_DIS
LIN {X -0.117,Y -377.389,Z 1595.612,A 0.000,B 0.000,C 90.000,E1 290.120} C_DIS
LIN {X -0.130,Y -386.504,Z 1595.605,A 0.000,B 0.000,C 90.000,E1 288.960} C_DIS
LIN {X 0.184,Y -392.795,Z 1595.600,A 0.000,B 0.000,C 90.000,E1 288.055} C_DIS
LIN {X 0.061,Y -398.515,Z 1595.596,A 0.000,B 0.000,C 90.000,E1 287.221} C_DIS
LIN {X -0.079,Y -402.018,Z 1595.593,A 0.000,B 0.000,C 90.000,E1 286.677} C_DIS
LIN {X -0.114,Y -406.513,Z 1595.588,A 0.000,B 0.000,C 90.000,E1 285.843} C_DIS
LIN {X -0.111,Y -410.096,Z 1595.583,A 0.000,B 0.000,C 90.000,E1 285.009} C_DIS
LIN {X 0.107,Y -411.987,Z 1595.580,A 0.000,B 0.000,C 90.000,E1 284.426} C_DIS
LIN {X 0.036,Y -413.472,Z 1595.577,A 0.000,B 0.000,C 90.000,E1 283.883} C_DIS
LIN {X -0.127,Y -414.569,Z 1595.574,A 0.000,B 0.000,C 90.000,E1 283.355} C_DIS
LIN {X 0.126,Y -415.194,Z 1595.571,A 0.000,B 0.000,C 90.000,E1 282.771} C_DIS
LIN {X -0.019,Y -415.331,Z 1595.568,A 0.000,B 0.000,C 90.000,E1 282.243} C_DIS
LIN {X -0.160,Y -415.033,Z 1595.565,A 0.000,B 0.000,C 90.000,E1 281.715} C_DIS
LIN {X 0.107,Y -414.176,Z 1595.562,A 0.000,B 0.000,C 90.000,E1 281.130} C_DIS
LIN {X -0.038,Y -412.780,Z 1595.559,A 0.000,B 0.000,C 90.000,E1 280.602} C_DIS
LIN {X 0.217,Y -410.734,Z 1595.556,A 0.000,B 0.000,C 90.000,E1 280.018} C_DIS
LIN {X -0.011,Y -408.058,Z 1595.553,A 0.000,B 0.000,C 90.000,E1 279.500} C_DIS
LIN {X -0.190,Y -404.625,Z 1595.550,A 0.000,B 0.000,C 90.000,E1 278.973} C_DIS
LIN {X -0.048,Y -400.527,Z 1595.547,A 0.000,B 0.000,C 90.000,E1 278.398} C_DIS
LIN {X 0.127,Y -395.669,Z 1595.543,A 0.000,B 0.000,C 90.000,E1 277.814} C_DIS
LIN {X -0.172,Y -390.176,Z 1595.540,A 0.000,B 0.000,C 90.000,E1 277.296} C_DIS
LIN {X 0.147,Y -384.377,Z 1595.537,A 0.000,B 0.000,C 90.000,E1 276.720} C_DIS
LIN {X -0.018,Y -378.422,Z 1595.535,A 0.000,B 0.000,C 90.000,E1 276.258} C_DIS
LIN {X 0.069,Y -372.196,Z 1595.532,A 0.000,B 0.000,C 90.000,E1 275.796} C_DIS
LIN {X 0.044,Y -365.926,Z 1595.530,A 0.000,B 0.000,C 90.000,E1 275.391} C_DIS
LIN {X -0.178,Y -359.513,Z 1595.528,A 0.000,B 0.000,C 90.000,E1 275.049} C_DIS
LIN {X -0.110,Y -349.708,Z 1595.525,A 0.000,B 0.000,C 90.000,E1 274.531} C_DIS
LIN {X -0.095,Y -339.920,Z 1595.523,A 0.000,B 0.000,C 90.000,E1 274.073} C_DIS
LIN {X -0.124,Y -330.184,Z 1595.520,A 0.000,B 0.000,C 90.000,E1 273.669} C_DIS
LIN {X -0.006,Y -320.270,Z 1595.518,A 0.000,B 0.000,C 90.000,E1 273.269} C_DIS
LIN {X 0.029,Y -310.147,Z 1595.516,A 0.000,B 0.000,C 90.000,E1 272.922} C_DIS
LIN {X -0.071,Y -299.271,Z 1595.515,A 0.000,B 0.000,C 90.000,E1 272.636} C_DIS
LIN {X -0.101,Y -287.998,Z 1595.513,A 0.000,B 0.000,C 90.000,E1 272.407} C_DIS
LIN {X 0.106,Y -274.105,Z 1595.512,A 0.000,B 0.000,C 90.000,E1 272.178} C_DIS
LIN {X -0.070,Y -260.738,Z 1595.511,A 0.000,B 0.000,C 90.000,E1 272.064} C_DIS
LIN {X -0.099,Y -244.899,Z 1595.511,A 0.000,B 0.000,C 90.000,E1 271.949} C_DIS
LIN {X -0.043,Y -233.694,Z 1595.510,A 0.000,B 0.000,C 90.000,E1 271.892} C_DIS
LIN {X -0.066,Y -181.284,Z 1595.510,A 0.000,B 0.000,C 90.000,E1 271.892} C_DIS
LIN {X 0.064,Y -181.576,Z 1595.501,A 0.000,B 0.000,C 90.000,E1 270.115} C_DIS
LIN {X 0.051,Y -180.878,Z 1595.473,A 0.000,B 0.000,C 90.000,E1 265.065} C_DIS
LIN {X -0.069,Y -178.996,Z 1595.445,A 0.000,B 0.000,C 90.000,E1 260.038} C_DIS
LIN {X 0.025,Y -178.585,Z 1595.440,A 0.000,B 0.000,C 90.000,E1 259.162} C_DIS
LIN {X -0.081,Y -175.637,Z 1595.411,A 0.000,B 0.000,C 90.000,E1 254.102} C_DIS
LIN {X -0.075,Y -172.357,Z 1595.388,A 0.000,B 0.000,C 90.000,E1 249.826} C_DIS
LIN {X -0.060,Y -171.143,Z 1595.378,A 0.000,B 0.000,C 90.000,E1 248.103} C_DIS
LIN {X -0.015,Y -167.447,Z 1595.354,A 0.000,B 0.000,C 90.000,E1 243.768} C_DIS
LIN {X 0.067,Y -166.843,Z 1595.349,A 0.000,B 0.000,C 90.000,E1 242.871} C_DIS
LIN {X -0.016,Y -162.826,Z 1595.325,A 0.000,B 0.000,C 90.000,E1 238.535} C_DIS
LIN {X 0.047,Y -161.511,Z 1595.315,A 0.000,B 0.000,C 90.000,E1 236.755} C_DIS
LIN {X 0.000,Y -157.509,Z 1595.291,A 0.000,B 0.000,C 90.000,E1 232.351} C_DIS
LIN {X 0.034,Y -155.531,Z 1595.276,A 0.000,B 0.000,C 90.000,E1 229.666} C_DIS
LIN {X 0.083,Y -151.827,Z 1595.251,A 0.000,B 0.000,C 90.000,E1 225.162} C_DIS
LIN {X -0.006,Y -150.044,Z 1595.236,A 0.000,B 0.000,C 90.000,E1 222.486} C_DIS
LIN {X 0.008,Y -146.859,Z 1595.211,A 0.000,B 0.000,C 90.000,E1 217.935} C_DIS
LIN {X 0.027,Y -145.443,Z 1595.196,A 0.000,B 0.000,C 90.000,E1 215.185} C_DIS
LIN {X 0.022,Y -142.863,Z 1595.170,A 0.000,B 0.000,C 90.000,E1 210.590} C_DIS
LIN {X 0.074,Y -141.479,Z 1595.149,A 0.000,B 0.000,C 90.000,E1 206.873} C_DIS
LIN {X -0.066,Y -139.381,Z 1595.113,A 0.000,B 0.000,C 90.000,E1 200.429} C_DIS
LIN {X 0.055,Y -138.835,Z 1595.098,A 0.000,B 0.000,C 90.000,E1 197.583} C_DIS
LIN {X -0.017,Y -138.353,Z 1595.056,A 0.000,B 0.000,C 90.000,E1 190.141} C_DIS
LIN {X -0.022,Y -139.524,Z 1595.004,A 0.000,B 0.000,C 90.000,E1 180.802} C_DIS
LIN {X 0.059,Y -141.193,Z 1594.973,A 0.000,B 0.000,C 90.000,E1 175.184} C_DIS
LIN {X 0.030,Y -142.569,Z 1594.958,A 0.000,B 0.000,C 90.000,E1 172.413} C_DIS
LIN {X -0.015,Y -144.857,Z 1594.932,A 0.000,B 0.000,C 90.000,E1 167.813} C_DIS
LIN {X -0.060,Y -147.482,Z 1594.912,A 0.000,B 0.000,C 90.000,E1 164.157} C_DIS
LIN {X -0.034,Y -150.068,Z 1594.892,A 0.000,B 0.000,C 90.000,E1 160.496} C_DIS
LIN {X -0.029,Y -153.417,Z 1594.871,A 0.000,B 0.000,C 90.000,E1 156.869} C_DIS
LIN {X 0.018,Y -156.837,Z 1594.851,A 0.000,B 0.000,C 90.000,E1 153.256} C_DIS
LIN {X 0.090,Y -160.916,Z 1594.832,A 0.000,B 0.000,C 90.000,E1 149.665} C_DIS
LIN {X 0.035,Y -163.041,Z 1594.822,A 0.000,B 0.000,C 90.000,E1 147.916} C_DIS
LIN {X 0.039,Y -167.433,Z 1594.802,A 0.000,B 0.000,C 90.000,E1 144.402} C_DIS
LIN {X -0.052,Y -171.271,Z 1594.788,A 0.000,B 0.000,C 90.000,E1 141.823} C_DIS
LIN {X -0.012,Y -176.163,Z 1594.769,A 0.000,B 0.000,C 90.000,E1 138.366} C_DIS
LIN {X -0.014,Y -180.434,Z 1594.755,A 0.000,B 0.000,C 90.000,E1 135.810} C_DIS
LIN {X -0.039,Y -185.840,Z 1594.736,A 0.000,B 0.000,C 90.000,E1 132.447} C_DIS
LIN {X 0.014,Y -190.462,Z 1594.722,A 0.000,B 0.000,C 90.000,E1 129.930} C_DIS
LIN {X -0.080,Y -196.214,Z 1594.704,A 0.000,B 0.000,C 90.000,E1 126.664} C_DIS
LIN {X -0.004,Y -201.024,Z 1594.690,A 0.000,B 0.000,C 90.000,E1 124.199} C_DIS
LIN {X -0.011,Y -204.802,Z 1594.678,A 0.000,B 0.000,C 90.000,E1 122.084} C_DIS
LIN {X -0.066,Y -322.997,Z 1594.678,A 0.000,B 0.000,C 90.000,E1 122.084} C_DIS
LIN {X -0.025,Y -327.640,Z 1594.677,A 0.000,B 0.000,C 90.000,E1 121.926} C_DIS
LIN {X -0.109,Y -329.830,Z 1594.677,A 0.000,B 0.000,C 90.000,E1 121.799} C_DIS
LIN {X 0.027,Y -333.713,Z 1594.674,A 0.000,B 0.000,C 90.000,E1 121.386} C_DIS
LIN {X -0.057,Y -337.139,Z 1594.671,A 0.000,B 0.000,C 90.000,E1 120.846} C_DIS
LIN {X -0.079,Y -351.657,Z 1594.652,A 0.000,B 0.000,C 90.000,E1 117.462} C_DIS
LIN {X -0.191,Y -365.031,Z 1594.637,A 0.000,B 0.000,C 90.000,E1 114.771} C_DIS
LIN {X 0.106,Y -379.966,Z 1594.623,A 0.000,B 0.000,C 90.000,E1 112.078} C_DIS
LIN {X -0.124,Y -394.662,Z 1594.610,A 0.000,B 0.000,C 90.000,E1 109.812} C_DIS
LIN {X 0.133,Y -410.797,Z 1594.598,A 0.000,B 0.000,C 90.000,E1 107.528} C_DIS
LIN {X -0.116,Y -428.484,Z 1594.585,A 0.000,B 0.000,C 90.000,E1 105.371} C_DIS
LIN {X -0.112,Y -447.768,Z 1594.573,A 0.000,B 0.000,C 90.000,E1 103.244} C_DIS
LIN {X 0.071,Y -467.896,Z 1594.563,A 0.000,B 0.000,C 90.000,E1 101.243} C_DIS
LIN {X 0.055,Y -491.183,Z 1594.551,A 0.000,B 0.000,C 90.000,E1 99.208} C_DIS
LIN {X -0.134,Y -496.214,Z 1594.549,A 0.000,B 0.000,C 90.000,E1 98.803} C_DIS
LIN {X -0.042,Y -498.128,Z 1594.548,A 0.000,B 0.000,C 90.000,E1 98.568} C_DIS
LIN {X -0.022,Y -499.587,Z 1594.546,A 0.000,B 0.000,C 90.000,E1 98.341} C_DIS
LIN {X -0.097,Y -500.784,Z 1594.545,A 0.000,B 0.000,C 90.000,E1 98.106} C_DIS
LIN {X -0.176,Y -501.650,Z 1594.544,A 0.000,B 0.000,C 90.000,E1 97.871} C_DIS
LIN {X 0.112,Y -502.538,Z 1594.541,A 0.000,B 0.000,C 90.000,E1 97.352} C_DIS
LIN {X -0.092,Y -502.416,Z 1594.538,A 0.000,B 0.000,C 90.000,E1 96.891} C_DIS
LIN {X 0.207,Y -501.263,Z 1594.536,A 0.000,B 0.000,C 90.000,E1 96.372} C_DIS
LIN {X 0.080,Y -500.246,Z 1594.534,A 0.000,B 0.000,C 90.000,E1 96.144} C_DIS
LIN {X 0.007,Y -498.866,Z 1594.533,A 0.000,B 0.000,C 90.000,E1 95.910} C_DIS
LIN {X -0.164,Y -484.050,Z 1594.521,A 0.000,B 0.000,C 90.000,E1 93.726} C_DIS
LIN {X -0.183,Y -474.084,Z 1594.512,A 0.000,B 0.000,C 90.000,E1 92.236} C_DIS
LIN {X -0.166,Y -465.517,Z 1594.505,A 0.000,B 0.000,C 90.000,E1 90.974} C_DIS
LIN {X -0.046,Y -454.712,Z 1594.497,A 0.000,B 0.000,C 90.000,E1 89.427} C_DIS
LIN {X 0.140,Y -445.299,Z 1594.490,A 0.000,B 0.000,C 90.000,E1 88.108} C_DIS
LIN {X 0.193,Y -435.441,Z 1594.482,A 0.000,B 0.000,C 90.000,E1 86.788} C_DIS
LIN {X -0.201,Y -423.310,Z 1594.473,A 0.000,B 0.000,C 90.000,E1 85.241} C_DIS
LIN {X 0.097,Y -403.827,Z 1594.458,A 0.000,B 0.000,C 90.000,E1 82.470} C_DIS
LIN {X -0.111,Y -385.793,Z 1594.443,A 0.000,B 0.000,C 90.000,E1 79.690} C_DIS
LIN {X 0.101,Y -368.825,Z 1594.427,A 0.000,B 0.000,C 90.000,E1 76.769} C_DIS
LIN {X 0.156,Y -355.819,Z 1594.413,A 0.000,B 0.000,C 90.000,E1 74.393} C_DIS
LIN {X 0.006,Y -343.129,Z 1594.400,A 0.000,B 0.000,C 90.000,E1 72.000} C_DIS
LIN {X 0.060,Y -329.342,Z 1594.385,A 0.000,B 0.000,C 90.000,E1 69.209} C_DIS
LIN {X 0.024,Y -314.880,Z 1594.367,A 0.000,B 0.000,C 90.000,E1 66.049} C_DIS
LIN {X 0.073,Y -301.503,Z 1594.349,A 0.000,B 0.000,C 90.000,E1 62.794} C_DIS
LIN {X 0.145,Y -293.531,Z 1594.338,A 0.000,B 0.000,C 90.000,E1 60.795} C_DIS
LIN {X 0.095,Y -285.214,Z 1594.327,A 0.000,B 0.000,C 90.000,E1 58.791} C_DIS
LIN {X 0.045,Y -276.438,Z 1594.315,A 0.000,B 0.000,C 90.000,E1 56.755} C_DIS
LIN {X -0.017,Y -267.548,Z 1594.304,A 0.000,B 0.000,C 90.000,E1 54.689} C_DIS
LIN {X 0.035,Y -254.665,Z 1594.286,A 0.000,B 0.000,C 90.000,E1 51.492} C_DIS
LIN {X -0.033,Y -242.850,Z 1594.268,A 0.000,B 0.000,C 90.000,E1 48.243} C_DIS
LIN {X 0.105,Y -233.274,Z 1594.251,A 0.000,B 0.000,C 90.000,E1 45.243} C_DIS
LIN {X 0.109,Y -223.422,Z 1594.233,A 0.000,B 0.000,C 90.000,E1 41.838} C_DIS
LIN {X 0.011,Y -215.453,Z 1594.215,A 0.000,B 0.000,C 90.000,E1 38.785} C_DIS
LIN {X 0.051,Y -208.209,Z 1594.198,A 0.000,B 0.000,C 90.000,E1 35.644} C_DIS
LIN {X 0.046,Y -201.770,Z 1594.180,A 0.000,B 0.000,C 90.000,E1 32.467} C_DIS
LIN {X -0.087,Y -196.091,Z 1594.163,A 0.000,B 0.000,C 90.000,E1 29.283} C_DIS
LIN {X 0.064,Y -191.189,Z 1594.144,A 0.000,B 0.000,C 90.000,E1 25.976} C_DIS
LIN {X 0.075,Y -185.963,Z 1594.121,A 0.000,B 0.000,C 90.000,E1 21.844} C_DIS
LIN {X 0.001,Y -181.630,Z 1594.098,A 0.000,B 0.000,C 90.000,E1 17.692} C_DIS
LIN {X -0.008,Y -178.078,Z 1594.075,A 0.000,B 0.000,C 90.000,E1 13.480} C_DIS
LIN {X -0.064,Y -174.920,Z 1594.047,A 0.000,B 0.000,C 90.000,E1 8.398} C_DIS
LIN {X -0.074,Y -172.518,Z 1594.013,A 0.000,B 0.000,C 90.000,E1 2.407} C_DIS
LIN {X -0.002,Y -173.300,Z 1593.935,A 0.000,B 0.000,C 90.000,E1 348.342} C_DIS
LIN {X 0.012,Y -176.065,Z 1593.907,A 0.000,B 0.000,C 90.000,E1 343.196} C_DIS
LIN {X -0.030,Y -179.691,Z 1593.883,A 0.000,B 0.000,C 90.000,E1 338.954} C_DIS
LIN {X 0.096,Y -183.491,Z 1593.864,A 0.000,B 0.000,C 90.000,E1 335.537} C_DIS
LIN {X -0.037,Y -188.018,Z 1593.846,A 0.000,B 0.000,C 90.000,E1 332.231} C_DIS
LIN {X -0.039,Y -193.276,Z 1593.827,A 0.000,B 0.000,C 90.000,E1 328.918} C_DIS
LIN {X -0.029,Y -199.301,Z 1593.809,A 0.000,B 0.000,C 90.000,E1 325.642} C_DIS
LIN {X 0.029,Y -206.064,Z 1593.791,A 0.000,B 0.000,C 90.000,E1 322.396} C_DIS
LIN {X 0.019,Y -213.726,Z 1593.773,A 0.000,B 0.000,C 90.000,E1 319.218} C_DIS
LIN {X -0.124,Y -222.321,Z 1593.756,A 0.000,B 0.000,C 90.000,E1 316.134} C_DIS
LIN {X 0.100,Y -231.811,Z 1593.739,A 0.000,B 0.000,C 90.000,E1 313.014} C_DIS
LIN {X 0.106,Y -242.466,Z 1593.722,A 0.000,B 0.000,C 90.000,E1 310.011} C_DIS
LIN {X 0.069,Y -248.563,Z 1593.714,A 0.000,B 0.000,C 90.000,E1 308.543} C_DIS
LIN {X -0.020,Y -257.120,Z 1593.704,A 0.000,B 0.000,C 90.000,E1 306.744} C_DIS
LIN {X 0.019,Y -266.805,Z 1593.694,A 0.000,B 0.000,C 90.000,E1 304.945} C_DIS
LIN {X 0.134,Y -277.351,Z 1593.684,A 0.000,B 0.000,C 90.000,E1 303.166} C_DIS
LIN {X -0.030,Y -296.009,Z 1593.669,A 0.000,B 0.000,C 90.000,E1 300.463} C_DIS
LIN {X -0.113,Y -310.977,Z 1593.658,A 0.000,B 0.000,C 90.000,E1 298.487} C_DIS
LIN {X -0.145,Y -323.378,Z 1593.649,A 0.000,B 0.000,C 90.000,E1 296.873} C_DIS
LIN {X -0.117,Y -335.722,Z 1593.640,A 0.000,B 0.000,C 90.000,E1 295.283} C_DIS
LIN {X 0.102,Y -347.777,Z 1593.632,A 0.000,B 0.000,C 90.000,E1 293.695} C_DIS
LIN {X 0.029,Y -365.093,Z 1593.620,A 0.000,B 0.000,C 90.000,E1 291.589} C_DIS
LIN {X -0.129,Y -374.983,Z 1593.613,A 0.000,B 0.000,C 90.000,E1 290.429} C_DIS
LIN {X 0.065,Y -382.054,Z 1593.609,A 0.000,B 0.000,C 90.000,E1 289.523} C_DIS
LIN {X -0.026,Y -388.689,Z 1593.604,A 0.000,B 0.000,C 90.000,E1 288.671} C_DIS
LIN {X -0.067,Y -394.872,Z 1593.599,A 0.000,B 0.000,C 90.000,E1 287.819} C_DIS
LIN {X -0.050,Y -400.441,Z 1593.594,A 0.000,B 0.000,C 90.000,E1 286.968} C_DIS
LIN {X 0.090,Y -403.770,Z 1593.591,A 0.000,B 0.000,C 90.000,E1 286.386} C_DIS
LIN {X -0.019,Y -406.704,Z 1593.588,A 0.000,B 0.000,C 90.000,E1 285.843} C_DIS
LIN {X -0.015,Y -410.309,Z 1593.583,A 0.000,B 0.000,C 90.000,E1 285.009} C_DIS
LIN {X -0.194,Y -412.225,Z 1593.580,A 0.000,B 0.000,C 90.000,E1 284.481} C_DIS
LIN {X 0.136,Y -413.765,Z 1593.577,A 0.000,B 0.000,C 90.000,E1 283.883} C_DIS
LIN {X -0.025,Y -414.888,Z 1593.574,A 0.000,B 0.000,C 90.000,E1 283.355} C_DIS
LIN {X -0.175,Y -415.523,Z 1593.571,A 0.000,B 0.000,C 90.000,E1 282.827} C_DIS
LIN {X 0.087,Y -415.715,Z 1593.568,A 0.000,B 0.000,C 90.000,E1 282.243} C_DIS
LIN {X -0.052,Y -415.417,Z 1593.565,A 0.000,B 0.000,C 90.000,E1 281.715} C_DIS
LIN {X -0.191,Y -414.599,Z 1593.562,A 0.000,B 0.000,C 90.000,E1 281.186} C_DIS
LIN {X 0.074,Y -413.233,Z 1593.559,A 0.000,B 0.000,C 90.000,E1 280.602} C_DIS
LIN {X -0.074,Y -411.284,Z 1593.556,A 0.000,B 0.000,C 90.000,E1 280.074} C_DIS
LIN {X 0.104,Y -408.616,Z 1593.553,A 0.000,B 0.000,C 90.000,E1 279.500} C_DIS
LIN {X -0.072,Y -405.239,Z 1593.550,A 0.000,B 0.000,C 90.000,E1 278.973} C_DIS
LIN {X 0.073,Y -401.190,Z 1593.547,A 0.000,B 0.000,C 90.000,E1 278.398} C_DIS
LIN {X -0.143,Y -396.358,Z 1593.544,A 0.000,B 0.000,C 90.000,E1 277.871} C_DIS
LIN {X -0.048,Y -390.835,Z 1593.541,A 0.000,B 0.000,C 90.000,E1 277.296} C_DIS
LIN {X -0.080,Y -385.124,Z 1593.538,A 0.000,B 0.000,C 90.000,E1 276.777} C_DIS
LIN {X 0.116,Y -379.131,Z 1593.535,A 0.000,B 0.000,C 90.000,E1 276.258} C_DIS
LIN {X 0.180,Y -372.827,Z 1593.532,A 0.000,B 0.000,C 90.000,E1 275.796} C_DIS
LIN {X 0.145,Y -366.484,Z 1593.530,A 0.000,B 0.000,C 90.000,E1 275.391} C_DIS
LIN {X -0.037,Y -360.176,Z 1593.528,A 0.000,B 0.000,C 90.000,E1 275.049} C_DIS
LIN {X 0.039,Y -350.509,Z 1593.525,A 0.000,B 0.000,C 90.000,E1 274.531} C_DIS
LIN {X 0.056,Y -340.723,Z 1593.523,A 0.000,B 0.000,C 90.000,E1 274.073} C_DIS
LIN {X -0.022,Y -327.894,Z 1593.520,A 0.000,B 0.000,C 90.000,E1 273.555} C_DIS
LIN {X -0.115,Y -318.177,Z 1593.518,A 0.000,B 0.000,C 90.000,E1 273.212} C_DIS
LIN {X -0.030,Y -308.098,Z 1593.516,A 0.000,B 0.000,C 90.000,E1 272.865} C_DIS
LIN {X -0.013,Y -297.432,Z 1593.514,A 0.000,B 0.000,C 90.000,E1 272.579} C_DIS
LIN {X 0.052,Y -289.532,Z 1593.513,A 0.000,B 0.000,C 90.000,E1 272.407} C_DIS
LIN {X -0.046,Y -276.049,Z 1593.512,A 0.000,B 0.000,C 90.000,E1 272.236} C_DIS
LIN {X 0.021,Y -262.568,Z 1593.511,A 0.000,B 0.000,C 90.000,E1 272.064} C_DIS
LIN {X -0.113,Y -243.425,Z 1593.511,A 0.000,B 0.000,C 90.000,E1 271.949} C_DIS
LIN {X -0.005,Y -234.834,Z 1593.510,A 0.000,B 0.000,C 90.000,E1 271.892} C_DIS
LIN {X -0.038,Y -181.282,Z 1593.510,A 0.000,B 0.000,C 90.000,E1 271.892} C_DIS
LIN {X -0.061,Y -181.578,Z 1593.501,A 0.000,B 0.000,C 90.000,E1 270.172} C_DIS
LIN {X -0.072,Y -180.881,Z 1593.473,A 0.000,B 0.000,C 90.000,E1 265.122} C_DIS
LIN {X -0.011,Y -179.001,Z 1593.445,A 0.000,B 0.000,C 90.000,E1 260.038} C_DIS
LIN {X 0.082,Y -178.598,Z 1593.440,A 0.000,B 0.000,C 90.000,E1 259.162} C_DIS
LIN {X -0.024,Y -175.650,Z 1593.412,A 0.000,B 0.000,C 90.000,E1 254.102} C_DIS
LIN {X -0.019,Y -172.369,Z 1593.388,A 0.000,B 0.000,C 90.000,E1 249.826} C_DIS
LIN {X -0.004,Y -171.161,Z 1593.378,A 0.000,B 0.000,C 90.000,E1 248.103} C_DIS
LIN {X 0.039,Y -167.460,Z 1593.354,A 0.000,B 0.000,C 90.000,E1 243.768} C_DIS
LIN {X -0.027,Y -166.857,Z 1593.349,A 0.000,B 0.000,C 90.000,E1 242.922} C_DIS
LIN {X 0.038,Y -162.841,Z 1593.325,A 0.000,B 0.000,C 90.000,E1 238.535} C_DIS
LIN {X 0.013,Y -161.524,Z 1593.316,A 0.000,B 0.000,C 90.000,E1 236.786} C_DIS
LIN {X 0.052,Y -157.525,Z 1593.291,A 0.000,B 0.000,C 90.000,E1 232.351} C_DIS
LIN {X -0.014,Y -155.549,Z 1593.276,A 0.000,B 0.000,C 90.000,E1 229.703} C_DIS
LIN {X -0.080,Y -151.841,Z 1593.251,A 0.000,B 0.000,C 90.000,E1 225.243} C_DIS
LIN {X -0.065,Y -150.060,Z 1593.236,A 0.000,B 0.000,C 90.000,E1 222.528} C_DIS
LIN {X -0.031,Y -146.870,Z 1593.211,A 0.000,B 0.000,C 90.000,E1 217.971} C_DIS
LIN {X -0.042,Y -145.455,Z 1593.196,A 0.000,B 0.000,C 90.000,E1 215.231} C_DIS
LIN {X 0.072,Y -142.872,Z 1593.170,A 0.000,B 0.000,C 90.000,E1 210.590} C_DIS
LIN {X -0.003,Y -141.489,Z 1593.150,A 0.000,B 0.000,C 90.000,E1 206.924} C_DIS
LIN {X -0.017,Y -139.384,Z 1593.113,A 0.000,B 0.000,C 90.000,E1 200.429} C_DIS
LIN {X -0.028,Y -138.840,Z 1593.098,A 0.000,B 0.000,C 90.000,E1 197.638} C_DIS
LIN {X 0.032,Y -138.354,Z 1593.056,A 0.000,B 0.000,C 90.000,E1 190.141} C_DIS
LIN {X 0.027,Y -139.521,Z 1593.005,A 0.000,B 0.000,C 90.000,E1 180.802} C_DIS
LIN {X -0.032,Y -141.183,Z 1592.974,A 0.000,B 0.000,C 90.000,E1 175.241} C_DIS
LIN {X -0.062,Y -142.562,Z 1592.958,A 0.000,B 0.000,C 90.000,E1 172.470} C_DIS
LIN {X 0.005,Y -144.844,Z 1592.932,A 0.000,B 0.000,C 90.000,E1 167.825} C_DIS
LIN {X -0.009,Y -147.468,Z 1592.912,A 0.000,B 0.000,C 90.000,E1 164.157} C_DIS
LIN {X 0.018,Y -150.053,Z 1592.892,A 0.000,B 0.000,C 90.000,E1 160.496} C_DIS
LIN {X 0.022,Y -153.397,Z 1592.872,A 0.000,B 0.000,C 90.000,E1 156.869} C_DIS
LIN {X 0.069,Y -155.927,Z 1592.857,A 0.000,B 0.000,C 90.000,E1 154.152} C_DIS
LIN {X 0.043,Y -159.794,Z 1592.837,A 0.000,B 0.000,C 90.000,E1 150.589} C_DIS
LIN {X 0.029,Y -162.035,Z 1592.827,A 0.000,B 0.000,C 90.000,E1 148.820} C_DIS
LIN {X 0.003,Y -166.229,Z 1592.807,A 0.000,B 0.000,C 90.000,E1 145.308} C_DIS
LIN {X 0.005,Y -171.246,Z 1592.788,A 0.000,B 0.000,C 90.000,E1 141.823} C_DIS
LIN {X -0.072,Y -176.134,Z 1592.769,A 0.000,B 0.000,C 90.000,E1 138.405} C_DIS
LIN {X 0.044,Y -180.402,Z 1592.755,A 0.000,B 0.000,C 90.000,E1 135.810} C_DIS
LIN {X 0.019,Y -185.808,Z 1592.736,A 0.000,B 0.000,C 90.000,E1 132.447} C_DIS
LIN {X 0.074,Y -190.427,Z 1592.722,A 0.000,B 0.000,C 90.000,E1 129.930} C_DIS
LIN {X -0.034,Y -197.752,Z 1592.699,A 0.000,B 0.000,C 90.000,E1 125.851} C_DIS
LIN {X 0.057,Y -200.994,Z 1592.690,A 0.000,B 0.000,C 90.000,E1 124.199} C_DIS
LIN {X -0.027,Y -204.719,Z 1592.678,A 0.000,B 0.000,C 90.000,E1 122.133} C_DIS
LIN {X -0.096,Y -322.350,Z 1592.678,A 0.000,B 0.000,C 90.000,E1 122.133} C_DIS
LIN {X -0.001,Y -327.528,Z 1592.677,A 0.000,B 0.000,C 90.000,E1 121.957} C_DIS
LIN {X -0.010,Y -329.917,Z 1592.677,A 0.000,B 0.000,C 90.000,E1 121.799} C_DIS
LIN {X 0.074,Y -333.767,Z 1592.674,A 0.000,B 0.000,C 90.000,E1 121.386} C_DIS
LIN {X -0.094,Y -335.673,Z 1592.673,A 0.000,B 0.000,C 90.000,E1 121.131} C_DIS
LIN {X -0.090,Y -337.173,Z 1592.671,A 0.000,B 0.000,C 90.000,E1 120.846} C_DIS
LIN {X -0.101,Y -351.650,Z 1592.652,A 0.000,B 0.000,C 90.000,E1 117.462} C_DIS
LIN {X 0.119,Y -365.026,Z 1592.637,A 0.000,B 0.000,C 90.000,E1 114.719} C_DIS
LIN {X 0.083,Y -379.965,Z 1592.623,A 0.000,B 0.000,C 90.000,E1 112.078} C_DIS
LIN {X -0.148,Y -394.661,Z 1592.610,A 0.000,B 0.000,C 90.000,E1 109.812} C_DIS
LIN {X 0.107,Y -410.799,Z 1592.597,A 0.000,B 0.000,C 90.000,E1 107.528} C_DIS
LIN {X -0.141,Y -428.487,Z 1592.585,A 0.000,B 0.000,C 90.000,E1 105.371} C_DIS
LIN {X -0.139,Y -447.773,Z 1592.573,A 0.000,B 0.000,C 90.000,E1 103.244} C_DIS
LIN {X 0.044,Y -467.902,Z 1592.563,A 0.000,B 0.000,C 90.000,E1 101.243} C_DIS
LIN {X 0.029,Y -491.190,Z 1592.551,A 0.000,B 0.000,C 90.000,E1 99.208} C_DIS
LIN {X -0.161,Y -496.188,Z 1592.549,A 0.000,B 0.000,C 90.000,E1 98.803} C_DIS
LIN {X -0.085,Y -498.087,Z 1592.547,A 0.000,B 0.000,C 90.000,E1 98.568} C_DIS
LIN {X -0.082,Y -499.533,Z 1592.546,A 0.000,B 0.000,C 90.000,E1 98.341} C_DIS
LIN {X 0.262,Y -501.552,Z 1592.544,A 0.000,B 0.000,C 90.000,E1 97.814} C_DIS
LIN {X 0.046,Y -502.408,Z 1592.541,A 0.000,B 0.000,C 90.000,E1 97.352} C_DIS
LIN {X -0.160,Y -502.251,Z 1592.538,A 0.000,B 0.000,C 90.000,E1 96.891} C_DIS
LIN {X 0.139,Y -501.062,Z 1592.536,A 0.000,B 0.000,C 90.000,E1 96.372} C_DIS
LIN {X 0.012,Y -500.021,Z 1592.534,A 0.000,B 0.000,C 90.000,E1 96.144} C_DIS
LIN {X -0.062,Y -498.615,Z 1592.533,A 0.000,B 0.000,C 90.000,E1 95.910} C_DIS
LIN {X -0.237,Y -483.816,Z 1592.521,A 0.000,B 0.000,C 90.000,E1 93.726} C_DIS
LIN {X 0.215,Y -473.862,Z 1592.512,A 0.000,B 0.000,C 90.000,E1 92.178} C_DIS
LIN {X 0.223,Y -465.309,Z 1592.505,A 0.000,B 0.000,C 90.000,E1 90.917} C_DIS
LIN {X -0.125,Y -454.508,Z 1592.497,A 0.000,B 0.000,C 90.000,E1 89.427} C_DIS
LIN {X 0.059,Y -445.101,Z 1592.490,A 0.000,B 0.000,C 90.000,E1 88.108} C_DIS
LIN {X 0.113,Y -435.235,Z 1592.482,A 0.000,B 0.000,C 90.000,E1 86.788} C_DIS
LIN {X 0.174,Y -423.120,Z 1592.473,A 0.000,B 0.000,C 90.000,E1 85.179} C_DIS
LIN {X 0.013,Y -403.644,Z 1592.458,A 0.000,B 0.000,C 90.000,E1 82.470} C_DIS
LIN {X 0.131,Y -387.376,Z 1592.444,A 0.000,B 0.000,C 90.000,E1 79.926} C_DIS
LIN {X 0.099,Y -368.660,Z 1592.427,A 0.000,B 0.000,C 90.000,E1 76.756} C_DIS
LIN {X 0.068,Y -355.672,Z 1592.413,A 0.000,B 0.000,C 90.000,E1 74.393} C_DIS
LIN {X -0.083,Y -342.975,Z 1592.400,A 0.000,B 0.000,C 90.000,E1 72.000} C_DIS
LIN {X -0.029,Y -329.181,Z 1592.385,A 0.000,B 0.000,C 90.000,E1 69.209} C_DIS
LIN {X 0.002,Y -316.132,Z 1592.369,A 0.000,B 0.000,C 90.000,E1 66.357} C_DIS
LIN {X -0.018,Y -301.253,Z 1592.349,A 0.000,B 0.000,C 90.000,E1 62.794} C_DIS
LIN {X 0.051,Y -293.248,Z 1592.338,A 0.000,B 0.000,C 90.000,E1 60.795} C_DIS
LIN {X -0.001,Y -284.904,Z 1592.327,A 0.000,B 0.000,C 90.000,E1 58.791} C_DIS
LIN {X -0.054,Y -276.120,Z 1592.315,A 0.000,B 0.000,C 90.000,E1 56.755} C_DIS
LIN {X -0.040,Y -265.794,Z 1592.302,A 0.000,B 0.000,C 90.000,E1 54.322} C_DIS
LIN {X 0.124,Y -253.119,Z 1592.284,A 0.000,B 0.000,C 90.000,E1 51.090} C_DIS
LIN {X 0.023,Y -241.474,Z 1592.266,A 0.000,B 0.000,C 90.000,E1 47.838} C_DIS
LIN {X -0.083,Y -230.913,Z 1592.247,A 0.000,B 0.000,C 90.000,E1 44.514} C_DIS
LIN {X 0.031,Y -221.288,Z 1592.228,A 0.000,B 0.000,C 90.000,E1 41.067} C_DIS
LIN {X 0.050,Y -213.511,Z 1592.211,A 0.000,B 0.000,C 90.000,E1 37.971} C_DIS
LIN {X 0.082,Y -206.525,Z 1592.194,A 0.000,B 0.000,C 90.000,E1 34.818} C_DIS
LIN {X -0.070,Y -200.265,Z 1592.176,A 0.000,B 0.000,C 90.000,E1 31.671} C_DIS
LIN {X -0.062,Y -194.830,Z 1592.158,A 0.000,B 0.000,C 90.000,E1 28.437} C_DIS
LIN {X -0.028,Y -190.140,Z 1592.140,A 0.000,B 0.000,C 90.000,E1 25.155} C_DIS
LIN {X -0.049,Y -185.115,Z 1592.117,A 0.000,B 0.000,C 90.000,E1 21.025} C_DIS
LIN {X 0.076,Y -180.979,Z 1592.094,A 0.000,B 0.000,C 90.000,E1 16.804} C_DIS
LIN {X 0.048,Y -177.606,Z 1592.070,A 0.000,B 0.000,C 90.000,E1 12.591} C_DIS
LIN {X -0.091,Y -174.678,Z 1592.042,A 0.000,B 0.000,C 90.000,E1 7.530} C_DIS
LIN {X 0.045,Y -172.461,Z 1592.008,A 0.000,B 0.000,C 90.000,E1 1.489} C_DIS
LIN {X 0.014,Y -173.522,Z 1591.935,A 0.000,B 0.000,C 90.000,E1 348.342} C_DIS
LIN {X 0.038,Y -176.314,Z 1591.907,A 0.000,B 0.000,C 90.000,E1 343.196} C_DIS
LIN {X 0.004,Y -179.923,Z 1591.883,A 0.000,B 0.000,C 90.000,E1 338.954} C_DIS
LIN {X 0.076,Y -184.770,Z 1591.860,A 0.000,B 0.000,C 90.000,E1 334.717} C_DIS
LIN {X 0.058,Y -189.473,Z 1591.841,A 0.000,B 0.000,C 90.000,E1 331.385} C_DIS
LIN {X -0.073,Y -194.892,Z 1591.823,A 0.000,B 0.000,C 90.000,E1 328.122} C_DIS
LIN {X -0.032,Y -201.058,Z 1591.805,A 0.000,B 0.000,C 90.000,E1 324.848} C_DIS
LIN {X 0.020,Y -207.998,Z 1591.787,A 0.000,B 0.000,C 90.000,E1 321.618} C_DIS
LIN {X 0.037,Y -215.865,Z 1591.769,A 0.000,B 0.000,C 90.000,E1 318.447} C_DIS
LIN {X 0.103,Y -224.620,Z 1591.752,A 0.000,B 0.000,C 90.000,E1 315.324} C_DIS
LIN {X 0.067,Y -234.321,Z 1591.735,A 0.000,B 0.000,C 90.000,E1 312.285} C_DIS
LIN {X -0.153,Y -242.393,Z 1591.723,A 0.000,B 0.000,C 90.000,E1 310.092} C_DIS
LIN {X -0.043,Y -248.448,Z 1591.714,A 0.000,B 0.000,C 90.000,E1 308.588} C_DIS
LIN {X 0.038,Y -255.192,Z 1591.706,A 0.000,B 0.000,C 90.000,E1 307.111} C_DIS
LIN {X 0.056,Y -264.645,Z 1591.696,A 0.000,B 0.000,C 90.000,E1 305.311} C_DIS
LIN {X -0.012,Y -277.170,Z 1591.684,A 0.000,B 0.000,C 90.000,E1 303.214} C_DIS
LIN {X 0.068,Y -293.403,Z 1591.671,A 0.000,B 0.000,C 90.000,E1 300.797} C_DIS
LIN {X -0.058,Y -308.323,Z 1591.660,A 0.000,B 0.000,C 90.000,E1 298.821} C_DIS
LIN {X 0.026,Y -320.777,Z 1591.651,A 0.000,B 0.000,C 90.000,E1 297.180} C_DIS
LIN {X 0.006,Y -333.126,Z 1591.642,A 0.000,B 0.000,C 90.000,E1 295.591} C_DIS
LIN {X 0.053,Y -345.245,Z 1591.634,A 0.000,B 0.000,C 90.000,E1 294.027} C_DIS
LIN {X 0.149,Y -362.434,Z 1591.622,A 0.000,B 0.000,C 90.000,E1 291.897} C_DIS
LIN {X 0.058,Y -374.836,Z 1591.614,A 0.000,B 0.000,C 90.000,E1 290.429} C_DIS
LIN {X 0.020,Y -384.243,Z 1591.607,A 0.000,B 0.000,C 90.000,E1 289.268} C_DIS
LIN {X -0.061,Y -390.805,Z 1591.602,A 0.000,B 0.000,C 90.000,E1 288.417} C_DIS
LIN {X -0.202,Y -396.828,Z 1591.598,A 0.000,B 0.000,C 90.000,E1 287.583} C_DIS
LIN {X 0.211,Y -402.277,Z 1591.593,A 0.000,B 0.000,C 90.000,E1 286.677} C_DIS
LIN {X 0.181,Y -406.868,Z 1591.588,A 0.000,B 0.000,C 90.000,E1 285.843} C_DIS
LIN {X 0.188,Y -410.477,Z 1591.583,A 0.000,B 0.000,C 90.000,E1 285.009} C_DIS
LIN {X 0.012,Y -412.452,Z 1591.580,A 0.000,B 0.000,C 90.000,E1 284.481} C_DIS
LIN {X -0.058,Y -414.015,Z 1591.577,A 0.000,B 0.000,C 90.000,E1 283.939} C_DIS
LIN {X 0.185,Y -415.162,Z 1591.574,A 0.000,B 0.000,C 90.000,E1 283.355} C_DIS
LIN {X 0.036,Y -415.877,Z 1591.571,A 0.000,B 0.000,C 90.000,E1 282.827} C_DIS
LIN {X -0.105,Y -416.078,Z 1591.568,A 0.000,B 0.000,C 90.000,E1 282.299} C_DIS
LIN {X 0.164,Y -415.838,Z 1591.565,A 0.000,B 0.000,C 90.000,E1 281.715} C_DIS
LIN {X 0.026,Y -415.051,Z 1591.562,A 0.000,B 0.000,C 90.000,E1 281.186} C_DIS
LIN {X -0.113,Y -413.757,Z 1591.559,A 0.000,B 0.000,C 90.000,E1 280.658} C_DIS
LIN {X 0.147,Y -411.842,Z 1591.556,A 0.000,B 0.000,C 90.000,E1 280.074} C_DIS
LIN {X -0.078,Y -409.237,Z 1591.553,A 0.000,B 0.000,C 90.000,E1 279.557} C_DIS
LIN {X 0.152,Y -405.905,Z 1591.550,A 0.000,B 0.000,C 90.000,E1 278.973} C_DIS
LIN {X -0.100,Y -401.913,Z 1591.547,A 0.000,B 0.000,C 90.000,E1 278.454} C_DIS
LIN {X 0.083,Y -397.189,Z 1591.544,A 0.000,B 0.000,C 90.000,E1 277.871} C_DIS
LIN {X 0.181,Y -391.718,Z 1591.541,A 0.000,B 0.000,C 90.000,E1 277.296} C_DIS
LIN {X 0.117,Y -385.921,Z 1591.538,A 0.000,B 0.000,C 90.000,E1 276.777} C_DIS
LIN {X -0.083,Y -379.955,Z 1591.535,A 0.000,B 0.000,C 90.000,E1 276.315} C_DIS
LIN {X -0.026,Y -373.639,Z 1591.532,A 0.000,B 0.000,C 90.000,E1 275.853} C_DIS
LIN {X -0.130,Y -364.237,Z 1591.529,A 0.000,B 0.000,C 90.000,E1 275.277} C_DIS
LIN {X 0.159,Y -354.563,Z 1591.526,A 0.000,B 0.000,C 90.000,E1 274.702} C_DIS
LIN {X 0.097,Y -344.950,Z 1591.524,A 0.000,B 0.000,C 90.000,E1 274.245} C_DIS
LIN {X -0.110,Y -332.062,Z 1591.521,A 0.000,B 0.000,C 90.000,E1 273.726} C_DIS
LIN {X 0.006,Y -319.000,Z 1591.518,A 0.000,B 0.000,C 90.000,E1 273.212} C_DIS
LIN {X 0.076,Y -308.916,Z 1591.516,A 0.000,B 0.000,C 90.000,E1 272.865} C_DIS
LIN {X 0.070,Y -298.170,Z 1591.514,A 0.000,B 0.000,C 90.000,E1 272.579} C_DIS
LIN {X 0.132,Y -290.264,Z 1591.514,A 0.000,B 0.000,C 90.000,E1 272.407} C_DIS
LIN {X 0.036,Y -277.120,Z 1591.512,A 0.000,B 0.000,C 90.000,E1 272.236} C_DIS
LIN {X 0.085,Y -263.726,Z 1591.512,A 0.000,B 0.000,C 90.000,E1 272.064} C_DIS
LIN {X -0.068,Y -244.534,Z 1591.511,A 0.000,B 0.000,C 90.000,E1 271.949} C_DIS
LIN {X 0.038,Y -235.656,Z 1591.511,A 0.000,B 0.000,C 90.000,E1 271.892} C_DIS
LIN {X -0.004,Y -181.280,Z 1591.510,A 0.000,B 0.000,C 90.000,E1 271.892} C_DIS
LIN {X -0.027,Y -181.578,Z 1591.501,A 0.000,B 0.000,C 90.000,E1 270.172} C_DIS
LIN {X -0.038,Y -180.883,Z 1591.473,A 0.000,B 0.000,C 90.000,E1 265.122} C_DIS
LIN {X 0.021,Y -179.003,Z 1591.445,A 0.000,B 0.000,C 90.000,E1 260.038} C_DIS
LIN {X -0.060,Y -178.606,Z 1591.440,A 0.000,B 0.000,C 90.000,E1 259.218} C_DIS
LIN {X 0.008,Y -175.658,Z 1591.412,A 0.000,B 0.000,C 90.000,E1 254.102} C_DIS
LIN {X 0.013,Y -172.376,Z 1591.388,A 0.000,B 0.000,C 90.000,E1 249.826} C_DIS
LIN {X 0.028,Y -171.172,Z 1591.378,A 0.000,B 0.000,C 90.000,E1 248.103} C_DIS
LIN {X 0.071,Y -167.468,Z 1591.354,A 0.000,B 0.000,C 90.000,E1 243.768} C_DIS
LIN {X 0.005,Y -166.864,Z 1591.350,A 0.000,B 0.000,C 90.000,E1 242.922} C_DIS
LIN {X 0.058,Y -162.168,Z 1591.320,A 0.000,B 0.000,C 90.000,E1 237.661} C_DIS
LIN {X -0.021,Y -160.730,Z 1591.311,A 0.000,B 0.000,C 90.000,E1 235.928} C_DIS
LIN {X -0.042,Y -157.534,Z 1591.291,A 0.000,B 0.000,C 90.000,E1 232.396} C_DIS
LIN {X 0.016,Y -155.560,Z 1591.276,A 0.000,B 0.000,C 90.000,E1 229.703} C_DIS
LIN {X -0.050,Y -151.850,Z 1591.251,A 0.000,B 0.000,C 90.000,E1 225.243} C_DIS
LIN {X -0.036,Y -150.069,Z 1591.236,A 0.000,B 0.000,C 90.000,E1 222.528} C_DIS
LIN {X -0.002,Y -146.876,Z 1591.211,A 0.000,B 0.000,C 90.000,E1 217.971} C_DIS
LIN {X -0.012,Y -145.462,Z 1591.196,A 0.000,B 0.000,C 90.000,E1 215.231} C_DIS
LIN {X -0.095,Y -142.877,Z 1591.170,A 0.000,B 0.000,C 90.000,E1 210.669} C_DIS
LIN {X 0.026,Y -141.494,Z 1591.150,A 0.000,B 0.000,C 90.000,E1 206.924} C_DIS
LIN {X 0.011,Y -139.386,Z 1591.114,A 0.000,B 0.000,C 90.000,E1 200.429} C_DIS
LIN {X -0.001,Y -138.843,Z 1591.098,A 0.000,B 0.000,C 90.000,E1 197.638} C_DIS
LIN {X 0.059,Y -138.354,Z 1591.057,A 0.000,B 0.000,C 90.000,E1 190.141} C_DIS
LIN {X 0.055,Y -139.519,Z 1591.005,A 0.000,B 0.000,C 90.000,E1 180.802} C_DIS
LIN {X -0.003,Y -141.178,Z 1590.974,A 0.000,B 0.000,C 90.000,E1 175.241} C_DIS
LIN {X -0.033,Y -142.557,Z 1590.958,A 0.000,B 0.000,C 90.000,E1 172.470} C_DIS
LIN {X 0.034,Y -144.836,Z 1590.932,A 0.000,B 0.000,C 90.000,E1 167.825} C_DIS
LIN {X 0.020,Y -147.460,Z 1590.912,A 0.000,B 0.000,C 90.000,E1 164.157} C_DIS
LIN {X 0.047,Y -150.044,Z 1590.892,A 0.000,B 0.000,C 90.000,E1 160.496} C_DIS
LIN {X 0.053,Y -153.385,Z 1590.872,A 0.000,B 0.000,C 90.000,E1 156.869} C_DIS
LIN {X -0.041,Y -155.916,Z 1590.857,A 0.000,B 0.000,C 90.000,E1 154.204} C_DIS
LIN {X 0.074,Y -159.781,Z 1590.837,A 0.000,B 0.000,C 90.000,E1 150.589} C_DIS
LIN {X -0.079,Y -162.020,Z 1590.827,A 0.000,B 0.000,C 90.000,E1 148.869} C_DIS
LIN {X 0.035,Y -166.215,Z 1590.807,A 0.000,B 0.000,C 90.000,E1 145.308} C_DIS
LIN {X 0.036,Y -171.231,Z 1590.788,A 0.000,B 0.000,C 90.000,E1 141.823} C_DIS
LIN {X -0.040,Y -176.117,Z 1590.769,A 0.000,B 0.000,C 90.000,E1 138.405} C_DIS
LIN {X 0.076,Y -180.382,Z 1590.755,A 0.000,B 0.000,C 90.000,E1 135.810} C_DIS
LIN {X 0.053,Y -185.790,Z 1590.736,A 0.000,B 0.000,C 90.000,E1 132.447} C_DIS
LIN {X -0.013,Y -190.407,Z 1590.722,A 0.000,B 0.000,C 90.000,E1 129.967} C_DIS
LIN {X 0.001,Y -197.731,Z 1590.699,A 0.000,B 0.000,C 90.000,E1 125.851} C_DIS
LIN {X 0.092,Y -200.977,Z 1590.690,A 0.000,B 0.000,C 90.000,E1 124.199} C_DIS
LIN {X 0.078,Y -204.664,Z 1590.679,A 0.000,B 0.000,C 90.000,E1 122.133} C_DIS
LIN {X 0.070,Y -322.801,Z 1590.679,A 0.000,B 0.000,C 90.000,E1 122.133} C_DIS
LIN {X -0.037,Y -323.878,Z 1590.678,A 0.000,B 0.000,C 90.000,E1 122.133} C_DIS
LIN {X 0.057,Y -327.834,Z 1590.678,A 0.000,B 0.000,C 90.000,E1 121.957} C_DIS
LIN {X 0.048,Y -330.090,Z 1590.677,A 0.000,B 0.000,C 90.000,E1 121.799} C_DIS
LIN {X 0.010,Y -333.962,Z 1590.674,A 0.000,B 0.000,C 90.000,E1 121.386} C_DIS
LIN {X 0.075,Y -335.838,Z 1590.673,A 0.000,B 0.000,C 90.000,E1 121.082} C_DIS
LIN {X 0.026,Y -337.312,Z 1590.671,A 0.000,B 0.000,C 90.000,E1 120.797} C_DIS
LIN {X 0.014,Y -350.367,Z 1590.654,A 0.000,B 0.000,C 90.000,E1 117.719} C_DIS
LIN {X -0.125,Y -363.589,Z 1590.639,A 0.000,B 0.000,C 90.000,E1 115.027} C_DIS
LIN {X 0.131,Y -378.368,Z 1590.624,A 0.000,B 0.000,C 90.000,E1 112.333} C_DIS
LIN {X -0.131,Y -392.909,Z 1590.611,A 0.000,B 0.000,C 90.000,E1 110.066} C_DIS
LIN {X -0.178,Y -408.878,Z 1590.599,A 0.000,B 0.000,C 90.000,E1 107.819} C_DIS
LIN {X -0.082,Y -426.385,Z 1590.587,A 0.000,B 0.000,C 90.000,E1 105.607} C_DIS
LIN {X -0.064,Y -445.523,Z 1590.575,A 0.000,B 0.000,C 90.000,E1 103.467} C_DIS
LIN {X -0.138,Y -465.589,Z 1590.564,A 0.000,B 0.000,C 90.000,E1 101.478} C_DIS
LIN {X 0.260,Y -488.786,Z 1590.552,A 0.000,B 0.000,C 90.000,E1 99.378} C_DIS
LIN {X 0.037,Y -494.027,Z 1590.550,A 0.000,B 0.000,C 90.000,E1 98.973} C_DIS
LIN {X 0.150,Y -496.328,Z 1590.549,A 0.000,B 0.000,C 90.000,E1 98.746} C_DIS
LIN {X 0.183,Y -498.193,Z 1590.547,A 0.000,B 0.000,C 90.000,E1 98.511} C_DIS
LIN {X 0.215,Y -499.609,Z 1590.546,A 0.000,B 0.000,C 90.000,E1 98.276} C_DIS
LIN {X -0.009,Y -501.521,Z 1590.543,A 0.000,B 0.000,C 90.000,E1 97.814} C_DIS
LIN {X -0.226,Y -502.290,Z 1590.541,A 0.000,B 0.000,C 90.000,E1 97.352} C_DIS
LIN {X 0.068,Y -502.053,Z 1590.538,A 0.000,B 0.000,C 90.000,E1 96.834} C_DIS
LIN {X -0.132,Y -500.773,Z 1590.535,A 0.000,B 0.000,C 90.000,E1 96.372} C_DIS
LIN {X -0.259,Y -499.679,Z 1590.534,A 0.000,B 0.000,C 90.000,E1 96.144} C_DIS
LIN {X 0.031,Y -496.523,Z 1590.531,A 0.000,B 0.000,C 90.000,E1 95.625} C_DIS
LIN {X -0.184,Y -481.800,Z 1590.519,A 0.000,B 0.000,C 90.000,E1 93.440} C_DIS
LIN {X -0.236,Y -471.801,Z 1590.511,A 0.000,B 0.000,C 90.000,E1 91.949} C_DIS
LIN {X 0.210,Y -463.162,Z 1590.504,A 0.000,B 0.000,C 90.000,E1 90.630} C_DIS
LIN {X 0.056,Y -454.152,Z 1590.497,A 0.000,B 0.000,C 90.000,E1 89.370} C_DIS
LIN {X -0.214,Y -444.723,Z 1590.489,A 0.000,B 0.000,C 90.000,E1 88.108} C_DIS
LIN {X -0.160,Y -434.841,Z 1590.482,A 0.000,B 0.000,C 90.000,E1 86.788} C_DIS
LIN {X -0.097,Y -422.731,Z 1590.473,A 0.000,B 0.000,C 90.000,E1 85.179} C_DIS
LIN {X 0.143,Y -403.281,Z 1590.458,A 0.000,B 0.000,C 90.000,E1 82.413} C_DIS
LIN {X -0.137,Y -387.044,Z 1590.444,A 0.000,B 0.000,C 90.000,E1 79.926} C_DIS
LIN {X 0.180,Y -366.703,Z 1590.425,A 0.000,B 0.000,C 90.000,E1 76.408} C_DIS
LIN {X 0.092,Y -353.772,Z 1590.411,A 0.000,B 0.000,C 90.000,E1 74.047} C_DIS
LIN {X -0.008,Y -341.097,Z 1590.398,A 0.000,B 0.000,C 90.000,E1 71.638} C_DIS
LIN {X -0.006,Y -327.403,Z 1590.382,A 0.000,B 0.000,C 90.000,E1 68.847} C_DIS
LIN {X 0.035,Y -315.836,Z 1590.368,A 0.000,B 0.000,C 90.000,E1 66.305} C_DIS
LIN {X -0.029,Y -302.234,Z 1590.350,A 0.000,B 0.000,C 90.000,E1 63.076} C_DIS
LIN {X -0.064,Y -294.197,Z 1590.339,A 0.000,B 0.000,C 90.000,E1 61.101} C_DIS
LIN {X 0.011,Y -285.861,Z 1590.328,A 0.000,B 0.000,C 90.000,E1 59.076} C_DIS
LIN {X 0.011,Y -278.630,Z 1590.319,A 0.000,B 0.000,C 90.000,E1 57.375} C_DIS
LIN {X -0.077,Y -268.354,Z 1590.305,A 0.000,B 0.000,C 90.000,E1 54.975} C_DIS
LIN {X -0.003,Y -255.545,Z 1590.288,A 0.000,B 0.000,C 90.000,E1 51.778} C_DIS
LIN {X -0.038,Y -243.711,Z 1590.270,A 0.000,B 0.000,C 90.000,E1 48.528} C_DIS
LIN {X 0.088,Y -232.967,Z 1590.251,A 0.000,B 0.000,C 90.000,E1 45.162} C_DIS
LIN {X 0.090,Y -223.167,Z 1590.232,A 0.000,B 0.000,C 90.000,E1 41.757} C_DIS
LIN {X -0.015,Y -215.259,Z 1590.215,A 0.000,B 0.000,C 90.000,E1 38.705} C_DIS
LIN {X -0.102,Y -208.087,Z 1590.198,A 0.000,B 0.000,C 90.000,E1 35.598} C_DIS
LIN {X -0.098,Y -201.699,Z 1590.180,A 0.000,B 0.000,C 90.000,E1 32.418} C_DIS
LIN {X 0.043,Y -196.088,Z 1590.162,A 0.000,B 0.000,C 90.000,E1 29.155} C_DIS
LIN {X 0.020,Y -191.253,Z 1590.144,A 0.000,B 0.000,C 90.000,E1 25.899} C_DIS
LIN {X 0.029,Y -186.102,Z 1590.121,A 0.000,B 0.000,C 90.000,E1 21.770} C_DIS
LIN {X 0.069,Y -181.841,Z 1590.098,A 0.000,B 0.000,C 90.000,E1 17.583} C_DIS
LIN {X -0.060,Y -178.317,Z 1590.074,A 0.000,B 0.000,C 90.000,E1 13.411} C_DIS
LIN {X 0.055,Y -175.243,Z 1590.046,A 0.000,B 0.000,C 90.000,E1 8.276} C_DIS
LIN {X 0.025,Y -173.145,Z 1590.018,A 0.000,B 0.000,C 90.000,E1 3.154} C_DIS
LIN {X 0.089,Y -174.135,Z 1589.931,A 0.000,B 0.000,C 90.000,E1 347.465} C_DIS
LIN {X 0.007,Y -177.186,Z 1589.902,A 0.000,B 0.000,C 90.000,E1 342.362} C_DIS
LIN {X 0.056,Y -181.052,Z 1589.878,A 0.000,B 0.000,C 90.000,E1 338.103} C_DIS
LIN {X 0.065,Y -186.091,Z 1589.855,A 0.000,B 0.000,C 90.000,E1 333.896} C_DIS
LIN {X -0.001,Y -190.975,Z 1589.837,A 0.000,B 0.000,C 90.000,E1 330.589} C_DIS
LIN {X 0.008,Y -196.501,Z 1589.818,A 0.000,B 0.000,C 90.000,E1 327.296} C_DIS
LIN {X -0.073,Y -202.865,Z 1589.800,A 0.000,B 0.000,C 90.000,E1 324.069} C_DIS
LIN {X -0.010,Y -209.982,Z 1589.782,A 0.000,B 0.000,C 90.000,E1 320.848} C_DIS
LIN {X -0.077,Y -218.036,Z 1589.765,A 0.000,B 0.000,C 90.000,E1 317.715} C_DIS
LIN {X 0.029,Y -226.936,Z 1589.748,A 0.000,B 0.000,C 90.000,E1 314.595} C_DIS
LIN {X -0.111,Y -236.894,Z 1589.731,A 0.000,B 0.000,C 90.000,E1 311.595} C_DIS
LIN {X -0.087,Y -243.765,Z 1589.721,A 0.000,B 0.000,C 90.000,E1 309.725} C_DIS
LIN {X 0.044,Y -249.953,Z 1589.712,A 0.000,B 0.000,C 90.000,E1 308.222} C_DIS
LIN {X -0.057,Y -256.881,Z 1589.704,A 0.000,B 0.000,C 90.000,E1 306.790} C_DIS
LIN {X 0.096,Y -268.535,Z 1589.692,A 0.000,B 0.000,C 90.000,E1 304.612} C_DIS
LIN {X -0.049,Y -281.492,Z 1589.681,A 0.000,B 0.000,C 90.000,E1 302.546} C_DIS
LIN {X 0.135,Y -298.184,Z 1589.667,A 0.000,B 0.000,C 90.000,E1 300.129} C_DIS
LIN {X 0.100,Y -313.169,Z 1589.656,A 0.000,B 0.000,C 90.000,E1 298.153} C_DIS
LIN {X -0.010,Y -327.739,Z 1589.646,A 0.000,B 0.000,C 90.000,E1 296.283} C_DIS
LIN {X -0.035,Y -337.575,Z 1589.639,A 0.000,B 0.000,C 90.000,E1 295.027} C_DIS
LIN {X -0.081,Y -359.597,Z 1589.624,A 0.000,B 0.000,C 90.000,E1 292.280} C_DIS
LIN {X -0.046,Y -372.026,Z 1589.615,A 0.000,B 0.000,C 90.000,E1 290.791} C_DIS
LIN {X -0.121,Y -381.684,Z 1589.609,A 0.000,B 0.000,C 90.000,E1 289.631} C_DIS
LIN {X -0.082,Y -390.628,Z 1589.603,A 0.000,B 0.000,C 90.000,E1 288.471} C_DIS
LIN {X 0.152,Y -396.718,Z 1589.598,A 0.000,B 0.000,C 90.000,E1 287.583} C_DIS
LIN {X 0.183,Y -402.232,Z 1589.593,A 0.000,B 0.000,C 90.000,E1 286.732} C_DIS
LIN {X 0.151,Y -406.849,Z 1589.589,A 0.000,B 0.000,C 90.000,E1 285.898} C_DIS
LIN {X -0.051,Y -409.446,Z 1589.585,A 0.000,B 0.000,C 90.000,E1 285.371} C_DIS
LIN {X -0.021,Y -412.600,Z 1589.581,A 0.000,B 0.000,C 90.000,E1 284.537} C_DIS
LIN {X -0.192,Y -414.219,Z 1589.578,A 0.000,B 0.000,C 90.000,E1 284.008} C_DIS
LIN {X 0.152,Y -415.405,Z 1589.575,A 0.000,B 0.000,C 90.000,E1 283.411} C_DIS
LIN {X 0.003,Y -416.181,Z 1589.572,A 0.000,B 0.000,C 90.000,E1 282.883} C_DIS
LIN {X -0.139,Y -416.478,Z 1589.568,A 0.000,B 0.000,C 90.000,E1 282.355} C_DIS
LIN {X 0.132,Y -416.285,Z 1589.566,A 0.000,B 0.000,C 90.000,E1 281.771} C_DIS
LIN {X -0.004,Y -415.570,Z 1589.563,A 0.000,B 0.000,C 90.000,E1 281.243} C_DIS
LIN {X -0.141,Y -414.328,Z 1589.559,A 0.000,B 0.000,C 90.000,E1 280.715} C_DIS
LIN {X 0.049,Y -412.479,Z 1589.556,A 0.000,B 0.000,C 90.000,E1 280.141} C_DIS
LIN {X -0.100,Y -409.957,Z 1589.553,A 0.000,B 0.000,C 90.000,E1 279.613} C_DIS
LIN {X 0.018,Y -408.477,Z 1589.552,A 0.000,B 0.000,C 90.000,E1 279.321} C_DIS
LIN {X 0.178,Y -404.903,Z 1589.549,A 0.000,B 0.000,C 90.000,E1 278.746} C_DIS
LIN {X -0.019,Y -400.593,Z 1589.546,A 0.000,B 0.000,C 90.000,E1 278.219} C_DIS
LIN {X 0.099,Y -395.564,Z 1589.543,A 0.000,B 0.000,C 90.000,E1 277.644} C_DIS
LIN {X -0.076,Y -389.972,Z 1589.540,A 0.000,B 0.000,C 90.000,E1 277.125} C_DIS
LIN {X -0.025,Y -384.164,Z 1589.537,A 0.000,B 0.000,C 90.000,E1 276.606} C_DIS
LIN {X -0.112,Y -378.037,Z 1589.534,A 0.000,B 0.000,C 90.000,E1 276.144} C_DIS
LIN {X 0.092,Y -371.734,Z 1589.532,A 0.000,B 0.000,C 90.000,E1 275.682} C_DIS
LIN {X 0.083,Y -362.190,Z 1589.528,A 0.000,B 0.000,C 90.000,E1 275.106} C_DIS
LIN {X 0.140,Y -352.560,Z 1589.526,A 0.000,B 0.000,C 90.000,E1 274.588} C_DIS
LIN {X 0.127,Y -342.741,Z 1589.523,A 0.000,B 0.000,C 90.000,E1 274.131} C_DIS
LIN {X 0.116,Y -333.242,Z 1589.521,A 0.000,B 0.000,C 90.000,E1 273.726} C_DIS
LIN {X -0.094,Y -320.251,Z 1589.518,A 0.000,B 0.000,C 90.000,E1 273.269} C_DIS
LIN {X -0.054,Y -310.132,Z 1589.516,A 0.000,B 0.000,C 90.000,E1 272.922} C_DIS
LIN {X -0.074,Y -299.462,Z 1589.515,A 0.000,B 0.000,C 90.000,E1 272.636} C_DIS
LIN {X -0.031,Y -291.584,Z 1589.514,A 0.000,B 0.000,C 90.000,E1 272.465} C_DIS
LIN {X -0.126,Y -274.339,Z 1589.512,A 0.000,B 0.000,C 90.000,E1 272.236} C_DIS
LIN {X -0.073,Y -260.038,Z 1589.511,A 0.000,B 0.000,C 90.000,E1 272.064} C_DIS
LIN {X -0.091,Y -242.251,Z 1589.511,A 0.000,B 0.000,C 90.000,E1 271.949} C_DIS
LIN {X 0.055,Y -233.438,Z 1589.511,A 0.000,B 0.000,C 90.000,E1 271.892} C_DIS
LIN {X 0.007,Y -181.279,Z 1589.510,A 0.000,B 0.000,C 90.000,E1 271.892} C_DIS
LIN {X 0.015,Y -181.579,Z 1589.501,A 0.000,B 0.000,C 90.000,E1 270.172} C_DIS
LIN {X 0.003,Y -180.886,Z 1589.473,A 0.000,B 0.000,C 90.000,E1 265.122} C_DIS
LIN {X 0.063,Y -179.007,Z 1589.445,A 0.000,B 0.000,C 90.000,E1 260.038} C_DIS
LIN {X -0.018,Y -178.615,Z 1589.440,A 0.000,B 0.000,C 90.000,E1 259.218} C_DIS
LIN {X 0.049,Y -175.667,Z 1589.412,A 0.000,B 0.000,C 90.000,E1 254.102} C_DIS
LIN {X 0.054,Y -172.384,Z 1589.388,A 0.000,B 0.000,C 90.000,E1 249.826} C_DIS
LIN {X 0.068,Y -171.185,Z 1589.378,A 0.000,B 0.000,C 90.000,E1 248.103} C_DIS
LIN {X -0.039,Y -167.477,Z 1589.354,A 0.000,B 0.000,C 90.000,E1 243.819} C_DIS
LIN {X -0.031,Y -166.874,Z 1589.350,A 0.000,B 0.000,C 90.000,E1 242.948} C_DIS
LIN {X -0.039,Y -162.178,Z 1589.321,A 0.000,B 0.000,C 90.000,E1 237.709} C_DIS
LIN {X 0.018,Y -160.745,Z 1589.311,A 0.000,B 0.000,C 90.000,E1 235.928} C_DIS
LIN {X -0.003,Y -157.544,Z 1589.291,A 0.000,B 0.000,C 90.000,E1 232.396} C_DIS
LIN {X -0.065,Y -155.572,Z 1589.276,A 0.000,B 0.000,C 90.000,E1 229.747} C_DIS
LIN {X -0.013,Y -151.859,Z 1589.251,A 0.000,B 0.000,C 90.000,E1 225.243} C_DIS
LIN {X 0.001,Y -150.081,Z 1589.236,A 0.000,B 0.000,C 90.000,E1 222.528} C_DIS
LIN {X 0.035,Y -146.885,Z 1589.211,A 0.000,B 0.000,C 90.000,E1 217.971} C_DIS
LIN {X 0.024,Y -145.471,Z 1589.196,A 0.000,B 0.000,C 90.000,E1 215.231} C_DIS
LIN {X -0.059,Y -142.883,Z 1589.170,A 0.000,B 0.000,C 90.000,E1 210.669} C_DIS
LIN {X -0.002,Y -141.502,Z 1589.150,A 0.000,B 0.000,C 90.000,E1 206.950} C_DIS
LIN {X 0.047,Y -139.389,Z 1589.114,A 0.000,B 0.000,C 90.000,E1 200.429} C_DIS
LIN {X 0.035,Y -138.845,Z 1589.098,A 0.000,B 0.000,C 90.000,E1 197.638} C_DIS
LIN {X -0.041,Y -138.353,Z 1589.057,A 0.000,B 0.000,C 90.000,E1 190.197} C_DIS
LIN {X -0.049,Y -139.517,Z 1589.005,A 0.000,B 0.000,C 90.000,E1 180.859} C_DIS
LIN {X 0.032,Y -141.172,Z 1588.974,A 0.000,B 0.000,C 90.000,E1 175.241} C_DIS
LIN {X 0.003,Y -142.551,Z 1588.958,A 0.000,B 0.000,C 90.000,E1 172.470} C_DIS
LIN {X -0.072,Y -144.828,Z 1588.932,A 0.000,B 0.000,C 90.000,E1 167.881} C_DIS
LIN {X 0.058,Y -147.450,Z 1588.912,A 0.000,B 0.000,C 90.000,E1 164.157} C_DIS
LIN {X -0.057,Y -150.032,Z 1588.892,A 0.000,B 0.000,C 90.000,E1 160.550} C_DIS
LIN {X -0.051,Y -153.370,Z 1588.872,A 0.000,B 0.000,C 90.000,E1 156.922} C_DIS
LIN {X -0.002,Y -155.903,Z 1588.857,A 0.000,B 0.000,C 90.000,E1 154.204} C_DIS
LIN {X -0.027,Y -159.764,Z 1588.837,A 0.000,B 0.000,C 90.000,E1 150.639} C_DIS
LIN {X -0.039,Y -162.003,Z 1588.827,A 0.000,B 0.000,C 90.000,E1 148.869} C_DIS
LIN {X 0.074,Y -166.197,Z 1588.807,A 0.000,B 0.000,C 90.000,E1 145.308} C_DIS
LIN {X 0.077,Y -171.212,Z 1588.788,A 0.000,B 0.000,C 90.000,E1 141.823} C_DIS
LIN {X 0.002,Y -176.096,Z 1588.769,A 0.000,B 0.000,C 90.000,E1 138.405} C_DIS
LIN {X 0.119,Y -180.358,Z 1588.755,A 0.000,B 0.000,C 90.000,E1 135.810} C_DIS
LIN {X 0.096,Y -185.767,Z 1588.736,A 0.000,B 0.000,C 90.000,E1 132.447} C_DIS
LIN {X 0.030,Y -190.382,Z 1588.722,A 0.000,B 0.000,C 90.000,E1 129.967} C_DIS
LIN {X -0.071,Y -197.706,Z 1588.699,A 0.000,B 0.000,C 90.000,E1 125.884} C_DIS
LIN {X -0.029,Y -200.955,Z 1588.690,A 0.000,B 0.000,C 90.000,E1 124.246} C_DIS
LIN {X -0.048,Y -204.582,Z 1588.679,A 0.000,B 0.000,C 90.000,E1 122.212} C_DIS
LIN {X -0.135,Y -321.551,Z 1588.679,A 0.000,B 0.000,C 90.000,E1 122.212} C_DIS
LIN {X -0.196,Y -322.767,Z 1588.679,A 0.000,B 0.000,C 90.000,E1 122.212} C_DIS
LIN {X -0.039,Y -327.711,Z 1588.678,A 0.000,B 0.000,C 90.000,E1 122.005} C_DIS
LIN {X 0.121,Y -330.183,Z 1588.677,A 0.000,B 0.000,C 90.000,E1 121.799} C_DIS
LIN {X 0.040,Y -334.015,Z 1588.674,A 0.000,B 0.000,C 90.000,E1 121.386} C_DIS
LIN {X 0.069,Y -335.879,Z 1588.673,A 0.000,B 0.000,C 90.000,E1 121.082} C_DIS
LIN {X -0.016,Y -337.338,Z 1588.671,A 0.000,B 0.000,C 90.000,E1 120.797} C_DIS
LIN {X -0.028,Y -350.377,Z 1588.654,A 0.000,B 0.000,C 90.000,E1 117.719} C_DIS
LIN {X -0.169,Y -363.603,Z 1588.639,A 0.000,B 0.000,C 90.000,E1 115.027} C_DIS
LIN {X 0.085,Y -378.385,Z 1588.624,A 0.000,B 0.000,C 90.000,E1 112.333} C_DIS
LIN {X -0.178,Y -392.929,Z 1588.611,A 0.000,B 0.000,C 90.000,E1 110.066} C_DIS
LIN {X 0.164,Y -408.903,Z 1588.599,A 0.000,B 0.000,C 90.000,E1 107.764} C_DIS
LIN {X -0.132,Y -426.414,Z 1588.587,A 0.000,B 0.000,C 90.000,E1 105.607} C_DIS
LIN {X -0.114,Y -445.556,Z 1588.575,A 0.000,B 0.000,C 90.000,E1 103.467} C_DIS
LIN {X -0.187,Y -465.624,Z 1588.564,A 0.000,B 0.000,C 90.000,E1 101.478} C_DIS
LIN {X 0.211,Y -488.824,Z 1588.552,A 0.000,B 0.000,C 90.000,E1 99.378} C_DIS
LIN {X -0.012,Y -494.065,Z 1588.550,A 0.000,B 0.000,C 90.000,E1 98.973} C_DIS
LIN {X 0.102,Y -496.320,Z 1588.549,A 0.000,B 0.000,C 90.000,E1 98.746} C_DIS
LIN {X 0.111,Y -498.171,Z 1588.547,A 0.000,B 0.000,C 90.000,E1 98.511} C_DIS
LIN {X 0.118,Y -499.572,Z 1588.546,A 0.000,B 0.000,C 90.000,E1 98.276} C_DIS
LIN {X -0.106,Y -501.433,Z 1588.543,A 0.000,B 0.000,C 90.000,E1 97.814} C_DIS
LIN {X 0.175,Y -502.161,Z 1588.541,A 0.000,B 0.000,C 90.000,E1 97.296} C_DIS
LIN {X -0.029,Y -501.884,Z 1588.538,A 0.000,B 0.000,C 90.000,E1 96.834} C_DIS
